LIN {X 0,Y 316.614,Z 405.184,A -85,B 0,C 180,E1 -15553.1,E2 -15553.1} C_VEL
LIN {X 0,Y 315.865,Z 416.609,A -85,B 0,C 180,E1 -15553.852,E2 -15553.852} C_VEL
LIN {X 0,Y 315.165,Z 425.435,A -85,B 0,C 180,E1 -15554.645,E2 -15554.645} C_VEL
LIN {X 0,Y 314.376,Z 433.849,A -85,B 0,C 180,E1 -15555.6,E2 -15555.6} C_VEL
LIN {X 0,Y 313.605,Z 441.806,A -85,B 0,C 180,E1 -15556.721,E2 -15556.721} C_VEL
LIN {X 0,Y 312.821,Z 449.237,A -85,B 0,C 180,E1 -15558.006,E2 -15558.006} C_VEL
LIN {X 0,Y 311.997,Z 456.768,A -85,B 0,C 180,E1 -15559.618,E2 -15559.618} C_VEL
LIN {X 0,Y 311.335,Z 463.636,A -85,B 0,C 180,E1 -15561.563,E2 -15561.563} C_VEL
LIN {X 0,Y 310.91,Z 468.838,A -85,B 0,C 180,E1 -15563.511,E2 -15563.511} C_VEL
LIN {X 0,Y 310.745,Z 472.647,A -85,B 0,C 180,E1 -15565.46,E2 -15565.46} C_VEL
LIN {X 0,Y 310.69,Z 475.122,A -85,B 0,C 180,E1 -15567.407,E2 -15567.407} C_VEL
LIN {X 0,Y 310.648,Z 476.084,A -85,B 0,C 180,E1 -15568.704,E2 -15568.704} C_VEL
LIN {X 0,Y 310.689,Z 476.502,A -85,B 0,C 180,E1 -15570,E2 -15570} C_VEL
LIN {X 0,Y 310.647,Z 476.448,A -85,B 0,C 180,E1 -15571.296,E2 -15571.296} C_VEL
LIN {X 0,Y 310.688,Z 475.928,A -85,B 0,C 180,E1 -15572.593,E2 -15572.593} C_VEL
LIN {X 0,Y 310.749,Z 474.907,A -85,B 0,C 180,E1 -15573.89,E2 -15573.89} C_VEL
LIN {X 0,Y 310.838,Z 472.302,A -85,B 0,C 180,E1 -15575.828,E2 -15575.828} C_VEL
LIN {X 0,Y 311.1,Z 469.9,A -85,B 0,C 180,E1 -15577.137,E2 -15577.137} C_VEL
LIN {X 0,Y 311.63,Z 465.034,A -85,B 0,C 180,E1 -15579.083,E2 -15579.083} C_VEL
LIN {X 0,Y 312.265,Z 459.797,A -85,B 0,C 180,E1 -15580.7,E2 -15580.7} C_VEL
LIN {X 0,Y 313.245,Z 453.258,A -85,B 0,C 180,E1 -15582.306,E2 -15582.306} C_VEL
LIN {X 0,Y 314.329,Z 445.108,A -85,B 0,C 180,E1 -15583.907,E2 -15583.907} C_VEL
LIN {X 0,Y 315.586,Z 435.56,A -85,B 0,C 180,E1 -15585.334,E2 -15585.334} C_VEL
LIN {X 0,Y 316.548,Z 427.654,A -85,B 0,C 180,E1 -15586.278,E2 -15586.278} C_VEL
LIN {X 0,Y 317.389,Z 419.536,A -85,B 0,C 180,E1 -15587.061,E2 -15587.061} C_VEL
LIN {X 0,Y 318.104,Z 411.379,A -85,B 0,C 180,E1 -15587.684,E2 -15587.684} C_VEL
LIN {X 0,Y 318.823,Z 401.925,A -85,B 0,C 180,E1 -15588.221,E2 -15588.221} C_VEL
LIN {X 0,Y 319.332,Z 392.463,A -85,B 0,C 180,E1 -15588.585,E2 -15588.585} C_VEL
LIN {X 0,Y 320.087,Z 349.277,A -85,B 0,C 180,E1 -15589.636,E2 -15589.636} C_VEL
LIN {X 0,Y 316.6,Z 326.517,A -85,B 0,C 180,E1 -15590.471,E2 -15590.471} C_VEL
LIN {X 0,Y 314.474,Z 315.593,A -85,B 0,C 180,E1 -15590.951,E2 -15590.951} C_VEL
LIN {X 0,Y 315.369,Z 306.754,A -85,B 0,C 180,E1 -15593.648,E2 -15593.648} C_VEL
LIN {X 0,Y 314.358,Z 300.169,A -85,B 0,C 180,E1 -15595.831,E2 -15595.831} C_VEL
LIN {X 0,Y 312.514,Z 291.37,A -85,B 0,C 180,E1 -15598.922,E2 -15598.922} C_VEL
LIN {X 0,Y 312.497,Z 291.374,A -85,B 0,C 180,E1 -15602.666,E2 -15602.666} C_VEL
LIN {X 0,Y 312.531,Z 291.369,A -85,B 0,C 180,E1 -15605.949,E2 -15605.949} C_VEL
LIN {X 0,Y 312.499,Z 291.376,A -85,B 0,C 180,E1 -15610.125,E2 -15610.125} C_VEL
LIN {X 0,Y 312.452,Z 291.381,A -85,B 0,C 180,E1 -15613.964,E2 -15613.964} C_VEL
LIN {X 0,Y 312.478,Z 291.372,A -85,B 0,C 180,E1 -15617.918,E2 -15617.918} C_VEL
LIN {X 0,Y 312.496,Z 291.372,A -85,B 0,C 180,E1 -15620.971,E2 -15620.971} C_VEL
LIN {X 0,Y 312.524,Z 291.367,A -85,B 0,C 180,E1 -15624.219,E2 -15624.219} C_VEL
LIN {X 0,Y 312.497,Z 291.363,A -85,B 0,C 180,E1 -15627.333,E2 -15627.333} C_VEL
LIN {X 0,Y 312.544,Z 291.363,A -85,B 0,C 180,E1 -15631.276,E2 -15631.276} C_VEL
LIN {X 0,Y 312.576,Z 291.359,A -85,B 0,C 180,E1 -15634.71,E2 -15634.71} C_VEL
LIN {X 0,Y 312.527,Z 291.357,A -85,B 0,C 180,E1 -15638.912,E2 -15638.912} C_VEL
LIN {X 0,Y 312.629,Z 291.354,A -85,B 0,C 180,E1 -15641.656,E2 -15641.656} C_VEL
LIN {X 0,Y 312.684,Z 291.339,A -85,B 0,C 180,E1 -15645.686,E2 -15645.686} C_VEL
LIN {X 0,Y 312.688,Z 291.339,A -85,B 0,C 180,E1 -15649.642,E2 -15649.642} C_VEL
LIN {X 0,Y 312.843,Z 291.319,A -85,B 0,C 180,E1 -15652.254,E2 -15652.254} C_VEL
LIN {X 0,Y 312.703,Z 291.34,A -85,B 0,C 180,E1 -15654.842,E2 -15654.842} C_VEL
LIN {X 0,Y 312.979,Z 291.306,A -85,B 0,C 180,E1 -15658.713,E2 -15658.713} C_VEL
LIN {X 0,Y 312.98,Z 291.301,A -85,B 0,C 180,E1 -15661.287,E2 -15661.287} C_VEL
LIN {X 0,Y 312.695,Z 291.348,A -85,B 0,C 180,E1 -15665.158,E2 -15665.158} C_VEL
LIN {X 0,Y 312.792,Z 291.324,A -85,B 0,C 180,E1 -15667.748,E2 -15667.748} C_VEL
LIN {X 0,Y 312.659,Z 291.344,A -85,B 0,C 180,E1 -15671.672,E2 -15671.672} C_VEL
LIN {X 0,Y 312.691,Z 291.348,A -85,B 0,C 180,E1 -15674.888,E2 -15674.888} C_VEL
LIN {X 0,Y 312.621,Z 291.36,A -85,B 0,C 180,E1 -15679.237,E2 -15679.237} C_VEL
LIN {X 0,Y 312.538,Z 291.368,A -85,B 0,C 180,E1 -15682.79,E2 -15682.79} C_VEL
LIN {X 0,Y 312.595,Z 291.36,A -85,B 0,C 180,E1 -15685.936,E2 -15685.936} C_VEL
LIN {X 0,Y 312.538,Z 291.366,A -85,B 0,C 180,E1 -15689.651,E2 -15689.651} C_VEL
LIN {X 0,Y 312.513,Z 291.372,A -85,B 0,C 180,E1 -15693.69,E2 -15693.69} C_VEL
LIN {X 0,Y 312.575,Z 291.364,A -85,B 0,C 180,E1 -15697.741,E2 -15697.741} C_VEL
LIN {X 0,Y 312.587,Z 291.595,A -85,B 0,C 180,E1 -15698.104,E2 -15698.104} C_VEL
LIN {X 0,Y 314.358,Z 300.158,A -85,B 0,C 180,E1 -15701.104,E2 -15701.104} C_VEL
LIN {X 0,Y 317.012,Z 307.823,A -85,B 0,C 180,E1 -15701.53,E2 -15701.53} C_VEL
LIN {X 0,Y 320.69,Z 326.341,A -85,B 0,C 180,E1 -15702.278,E2 -15702.278} C_VEL
LIN {X 0,Y 319.477,Z 377.531,A -85,B 0,C 180,E1 -15703.511,E2 -15703.511} C_VEL
LIN {X 0,Y 318.939,Z 388.047,A -85,B 0,C 180,E1 -15703.952,E2 -15703.952} C_VEL
LIN {X 0,Y 318.259,Z 399.5,A -85,B 0,C 180,E1 -15704.703,E2 -15704.703} C_VEL
LIN {X 0,Y 317.369,Z 408.898,A -85,B 0,C 180,E1 -15705.549,E2 -15705.549} C_VEL
LIN {X 0,Y 316.493,Z 417.2,A -85,B 0,C 180,E1 -15706.5,E2 -15706.5} C_VEL
LIN {X 0,Y 315.629,Z 424.127,A -85,B 0,C 180,E1 -15707.465,E2 -15707.465} C_VEL
LIN {X 0,Y 314.701,Z 430.774,A -85,B 0,C 180,E1 -15708.58,E2 -15708.58} C_VEL
LIN {X 0,Y 313.776,Z 437.342,A -85,B 0,C 180,E1 -15709.925,E2 -15709.925} C_VEL
LIN {X 0,Y 313.144,Z 441.993,A -85,B 0,C 180,E1 -15711.068,E2 -15711.068} C_VEL
LIN {X 0,Y 312.365,Z 447.101,A -85,B 0,C 180,E1 -15712.594,E2 -15712.594} C_VEL
LIN {X 0,Y 311.798,Z 451.176,A -85,B 0,C 180,E1 -15714.124,E2 -15714.124} C_VEL
LIN {X 0,Y 311.31,Z 454.327,A -85,B 0,C 180,E1 -15715.641,E2 -15715.641} C_VEL
LIN {X 0,Y 311.064,Z 456.676,A -85,B 0,C 180,E1 -15717.165,E2 -15717.165} C_VEL
LIN {X 0,Y 310.646,Z 458.729,A -85,B 0,C 180,E1 -15719.284,E2 -15719.284} C_VEL
LIN {X 0,Y 310.448,Z 459.46,A -85,B 0,C 180,E1 -15721.615,E2 -15721.615} C_VEL
LIN {X 0,Y 310.449,Z 459.064,A -85,B 0,C 180,E1 -15723.08,E2 -15723.08} C_VEL
LIN {X 0,Y 310.596,Z 457.727,A -85,B 0,C 180,E1 -15724.837,E2 -15724.837} C_VEL
LIN {X 0,Y 310.899,Z 455.22,A -85,B 0,C 180,E1 -15726.698,E2 -15726.698} C_VEL
LIN {X 0,Y 311.215,Z 452.076,A -85,B 0,C 180,E1 -15728.332,E2 -15728.332} C_VEL
LIN {X 0,Y 311.607,Z 448.166,A -85,B 0,C 180,E1 -15729.883,E2 -15729.883} C_VEL
LIN {X 0,Y 312.175,Z 442.501,A -85,B 0,C 180,E1 -15731.629,E2 -15731.629} C_VEL
LIN {X 0,Y 312.802,Z 436.87,A -85,B 0,C 180,E1 -15733.018,E2 -15733.018} C_VEL
LIN {X 0,Y 313.534,Z 430.031,A -85,B 0,C 180,E1 -15734.397,E2 -15734.397} C_VEL
LIN {X 0,Y 314.41,Z 421.641,A -85,B 0,C 180,E1 -15735.766,E2 -15735.766} C_VEL
LIN {X 0,Y 315.327,Z 412.215,A -85,B 0,C 180,E1 -15736.958,E2 -15736.958} C_VEL
LIN {X 0,Y 316.046,Z 403.63,A -85,B 0,C 180,E1 -15737.814,E2 -15737.814} C_VEL
LIN {X 0,Y 316.594,Z 394.035,A -85,B 0,C 180,E1 -15738.557,E2 -15738.557} C_VEL
LIN {X 0,Y 317.053,Z 384.456,A -85,B 0,C 180,E1 -15739.1,E2 -15739.1} C_VEL
LIN {X 0,Y 317.454,Z 374.313,A -85,B 0,C 180,E1 -15739.477,E2 -15739.477} C_VEL
LIN {X 0,Y 318.284,Z 325.044,A -85,B 0,C 180,E1 -15740.639,E2 -15740.639} C_VEL
LIN {X 0,Y 313.875,Z 300.254,A -85,B 0,C 180,E1 -15741.51,E2 -15741.51} C_VEL
LIN {X 0,Y 313.394,Z 294.514,A -85,B 0,C 180,E1 -15743.562,E2 -15743.562} C_VEL
LIN {X 0,Y 312.735,Z 291.343,A -85,B 0,C 180,E1 -15744.762,E2 -15744.762} C_VEL
LIN {X 0,Y 312.99,Z 291.307,A -85,B 0,C 180,E1 -15748.713,E2 -15748.713} C_VEL
LIN {X 0,Y 312.991,Z 291.307,A -85,B 0,C 180,E1 -15751.287,E2 -15751.287} C_VEL
LIN {X 0,Y 312.709,Z 291.341,A -85,B 0,C 180,E1 -15755.158,E2 -15755.158} C_VEL
LIN {X 0,Y 312.82,Z 291.33,A -85,B 0,C 180,E1 -15757.747,E2 -15757.747} C_VEL
LIN {X 0,Y 312.671,Z 291.346,A -85,B 0,C 180,E1 -15761.671,E2 -15761.671} C_VEL
LIN {X 0,Y 312.668,Z 291.349,A -85,B 0,C 180,E1 -15764.865,E2 -15764.865} C_VEL
LIN {X 0,Y 312.586,Z 291.357,A -85,B 0,C 180,E1 -15769.212,E2 -15769.212} C_VEL
LIN {X 0,Y 312.526,Z 291.369,A -85,B 0,C 180,E1 -15772.78,E2 -15772.78} C_VEL
LIN {X 0,Y 312.596,Z 291.356,A -85,B 0,C 180,E1 -15775.933,E2 -15775.933} C_VEL
LIN {X 0,Y 312.544,Z 291.363,A -85,B 0,C 180,E1 -15779.649,E2 -15779.649} C_VEL
LIN {X 0,Y 312.517,Z 291.366,A -85,B 0,C 180,E1 -15783.688,E2 -15783.688} C_VEL
LIN {X 0,Y 312.517,Z 291.37,A -85,B 0,C 180,E1 -15787.385,E2 -15787.385} C_VEL
LIN {X 0,Y 312.487,Z 291.369,A -85,B 0,C 180,E1 -15790.708,E2 -15790.708} C_VEL
LIN {X 0,Y 312.506,Z 291.367,A -85,B 0,C 180,E1 -15794.198,E2 -15794.198} C_VEL
LIN {X 0,Y 312.544,Z 291.365,A -85,B 0,C 180,E1 -15797.905,E2 -15797.905} C_VEL
LIN {X 0,Y 312.538,Z 291.366,A -85,B 0,C 180,E1 -15801.907,E2 -15801.907} C_VEL
LIN {X 0,Y 312.5,Z 291.37,A -85,B 0,C 180,E1 -15805.789,E2 -15805.789} C_VEL
LIN {X 0,Y 312.502,Z 291.369,A -85,B 0,C 180,E1 -15805.999,E2 -15805.999} C_VEL
LIN {X 0,Y 311.861,Z 291.447,A -85,B 0,C 180,E1 -15807.075,E2 -15807.075} C_VEL
LIN {X 0,Y 309.03,Z 291.799,A -85,B 0,C 180,E1 -15808.827,E2 -15808.827} C_VEL
LIN {X 0,Y 306.614,Z 292.105,A -85,B 0,C 180,E1 -15810.247,E2 -15810.247} C_VEL
LIN {X 0,Y 305.574,Z 292.231,A -85,B 0,C 180,E1 -15811.347,E2 -15811.347} C_VEL
LIN {X 0,Y 305.489,Z 292.238,A -85,B 0,C 180,E1 -15811.72,E2 -15811.72} C_VEL
LIN {X 0,Y 305.564,Z 292.236,A -85,B 0,C 180,E1 -15814.087,E2 -15814.087} C_VEL
LIN {X 0,Y 305.492,Z 292.242,A -85,B 0,C 180,E1 -15818.402,E2 -15818.402} C_VEL
LIN {X 0,Y 305.582,Z 292.228,A -85,B 0,C 180,E1 -15821.217,E2 -15821.217} C_VEL
LIN {X 0,Y 305.64,Z 292.222,A -85,B 0,C 180,E1 -15825.348,E2 -15825.348} C_VEL
LIN {X 0,Y 305.626,Z 292.224,A -85,B 0,C 180,E1 -15829.399,E2 -15829.399} C_VEL
LIN {X 0,Y 305.787,Z 292.203,A -85,B 0,C 180,E1 -15832.074,E2 -15832.074} C_VEL
LIN {X 0,Y 305.676,Z 292.219,A -85,B 0,C 180,E1 -15834.723,E2 -15834.723} C_VEL
LIN {X 0,Y 305.947,Z 292.185,A -85,B 0,C 180,E1 -15838.684,E2 -15838.684} C_VEL
LIN {X 0,Y 305.949,Z 292.188,A -85,B 0,C 180,E1 -15841.316,E2 -15841.316} C_VEL
LIN {X 0,Y 305.832,Z 292.198,A -85,B 0,C 180,E1 -15846.598,E2 -15846.598} C_VEL
LIN {X 0,Y 305.696,Z 292.217,A -85,B 0,C 180,E1 -15849.261,E2 -15849.261} C_VEL
LIN {X 0,Y 305.581,Z 292.232,A -85,B 0,C 180,E1 -15853.296,E2 -15853.296} C_VEL
LIN {X 0,Y 305.585,Z 292.232,A -85,B 0,C 180,E1 -15856.02,E2 -15856.02} C_VEL
LIN {X 0,Y 305.552,Z 292.235,A -85,B 0,C 180,E1 -15859.436,E2 -15859.436} C_VEL
LIN {X 0,Y 305.478,Z 292.241,A -85,B 0,C 180,E1 -15863.04,E2 -15863.04} C_VEL
LIN {X 0,Y 305.523,Z 292.241,A -85,B 0,C 180,E1 -15866.221,E2 -15866.221} C_VEL
LIN {X 0,Y 305.48,Z 292.241,A -85,B 0,C 180,E1 -15869.048,E2 -15869.048} C_VEL
LIN {X 0,Y 305.434,Z 292.25,A -85,B 0,C 180,E1 -15871.953,E2 -15871.953} C_VEL
LIN {X 0,Y 305.455,Z 292.246,A -85,B 0,C 180,E1 -15875.114,E2 -15875.114} C_VEL
LIN {X 0,Y 305.442,Z 292.25,A -85,B 0,C 180,E1 -15878.529,E2 -15878.529} C_VEL
LIN {X 0,Y 305.453,Z 292.248,A -85,B 0,C 180,E1 -15882.587,E2 -15882.587} C_VEL
LIN {X 0,Y 305.437,Z 292.25,A -85,B 0,C 180,E1 -15886.349,E2 -15886.349} C_VEL
LIN {X 0,Y 305.453,Z 292.245,A -85,B 0,C 180,E1 -15889.893,E2 -15889.893} C_VEL
LIN {X 0,Y 305.476,Z 292.244,A -85,B 0,C 180,E1 -15893.633,E2 -15893.633} C_VEL
LIN {X 0,Y 305.461,Z 292.245,A -85,B 0,C 180,E1 -15896.484,E2 -15896.484} C_VEL
LIN {X 0,Y 305.428,Z 292.252,A -85,B 0,C 180,E1 -15899.588,E2 -15899.588} C_VEL
LIN {X 0,Y 305.523,Z 292.28,A -85,B 0,C 180,E1 -15902.052,E2 -15902.052} C_VEL
LIN {X 0,Y 307.662,Z 303.716,A -85,B 0,C 180,E1 -15906.026,E2 -15906.026} C_VEL
LIN {X 0,Y 307.694,Z 307.146,A -85,B 0,C 180,E1 -15907.152,E2 -15907.152} C_VEL
LIN {X 0,Y 306.626,Z 316.497,A -85,B 0,C 180,E1 -15910.125,E2 -15910.125} C_VEL
LIN {X 0,Y 311.183,Z 350.857,A -85,B 0,C 180,E1 -15911.24,E2 -15911.24} C_VEL
LIN {X 0,Y 310.4,Z 393.592,A -85,B 0,C 180,E1 -15912.292,E2 -15912.292} C_VEL
LIN {X 0,Y 309.872,Z 403.563,A -85,B 0,C 180,E1 -15912.705,E2 -15912.705} C_VEL
LIN {X 0,Y 309.112,Z 414.767,A -85,B 0,C 180,E1 -15913.404,E2 -15913.404} C_VEL
LIN {X 0,Y 308.293,Z 424.721,A -85,B 0,C 180,E1 -15914.294,E2 -15914.294} C_VEL
LIN {X 0,Y 307.452,Z 433.226,A -85,B 0,C 180,E1 -15915.268,E2 -15915.268} C_VEL
LIN {X 0,Y 306.613,Z 441.254,A -85,B 0,C 180,E1 -15916.412,E2 -15916.412} C_VEL
LIN {X 0,Y 306.013,Z 447.028,A -85,B 0,C 180,E1 -15917.398,E2 -15917.398} C_VEL
LIN {X 0,Y 305.307,Z 453.471,A -85,B 0,C 180,E1 -15918.717,E2 -15918.717} C_VEL
LIN {X 0,Y 304.738,Z 458.821,A -85,B 0,C 180,E1 -15920.04,E2 -15920.04} C_VEL
LIN {X 0,Y 304.306,Z 463.278,A -85,B 0,C 180,E1 -15921.366,E2 -15921.366} C_VEL
LIN {X 0,Y 303.844,Z 468.514,A -85,B 0,C 180,E1 -15923.359,E2 -15923.359} C_VEL
LIN {X 0,Y 303.651,Z 472.353,A -85,B 0,C 180,E1 -15925.354,E2 -15925.354} C_VEL
LIN {X 0,Y 303.615,Z 474.879,A -85,B 0,C 180,E1 -15927.347,E2 -15927.347} C_VEL
LIN {X 0,Y 303.566,Z 475.848,A -85,B 0,C 180,E1 -15928.673,E2 -15928.673} C_VEL
LIN {X 0,Y 303.601,Z 476.291,A -85,B 0,C 180,E1 -15930,E2 -15930} C_VEL
LIN {X 0,Y 303.565,Z 476.263,A -85,B 0,C 180,E1 -15931.327,E2 -15931.327} C_VEL
LIN {X 0,Y 303.614,Z 475.769,A -85,B 0,C 180,E1 -15932.653,E2 -15932.653} C_VEL
LIN {X 0,Y 303.665,Z 474.758,A -85,B 0,C 180,E1 -15933.981,E2 -15933.981} C_VEL
LIN {X 0,Y 303.73,Z 472.564,A -85,B 0,C 180,E1 -15935.747,E2 -15935.747} C_VEL
LIN {X 0,Y 304.046,Z 469.815,A -85,B 0,C 180,E1 -15937.304,E2 -15937.304} C_VEL
LIN {X 0,Y 304.618,Z 465.004,A -85,B 0,C 180,E1 -15939.294,E2 -15939.294} C_VEL
LIN {X 0,Y 305.284,Z 459.813,A -85,B 0,C 180,E1 -15940.948,E2 -15940.948} C_VEL
LIN {X 0,Y 306.076,Z 454.747,A -85,B 0,C 180,E1 -15942.262,E2 -15942.262} C_VEL
LIN {X 0,Y 306.992,Z 448.655,A -85,B 0,C 180,E1 -15943.571,E2 -15943.571} C_VEL
LIN {X 0,Y 307.963,Z 441.26,A -85,B 0,C 180,E1 -15944.876,E2 -15944.876} C_VEL
LIN {X 0,Y 309.083,Z 433.349,A -85,B 0,C 180,E1 -15946.003,E2 -15946.003} C_VEL
LIN {X 0,Y 310.326,Z 423.508,A -85,B 0,C 180,E1 -15947.122,E2 -15947.122} C_VEL
LIN {X 0,Y 311.38,Z 412.054,A -85,B 0,C 180,E1 -15948.079,E2 -15948.079} C_VEL
LIN {X 0,Y 312.138,Z 402.465,A -85,B 0,C 180,E1 -15948.649,E2 -15948.649} C_VEL
LIN {X 0,Y 312.702,Z 392.836,A -85,B 0,C 180,E1 -15949.037,E2 -15949.037} C_VEL
LIN {X 0,Y 313.516,Z 350.323,A -85,B 0,C 180,E1 -15950.099,E2 -15950.099} C_VEL
LIN {X 0,Y 310.134,Z 327.944,A -85,B 0,C 180,E1 -15950.947,E2 -15950.947} C_VEL
LIN {X 0,Y 307.65,Z 315.355,A -85,B 0,C 180,E1 -15951.526,E2 -15951.526} C_VEL
LIN {X 0,Y 308.449,Z 307.895,A -85,B 0,C 180,E1 -15953.855,E2 -15953.855} C_VEL
LIN {X 0,Y 307.261,Z 300.885,A -85,B 0,C 180,E1 -15956.247,E2 -15956.247} C_VEL
LIN {X 0,Y 305.468,Z 292.248,A -85,B 0,C 180,E1 -15959.379,E2 -15959.379} C_VEL
LIN {X 0,Y 305.461,Z 292.248,A -85,B 0,C 180,E1 -15963.516,E2 -15963.516} C_VEL
LIN {X 0,Y 305.471,Z 292.249,A -85,B 0,C 180,E1 -15966.739,E2 -15966.739} C_VEL
LIN {X 0,Y 305.45,Z 292.256,A -85,B 0,C 180,E1 -15970.599,E2 -15970.599} C_VEL
LIN {X 0,Y 305.42,Z 292.259,A -85,B 0,C 180,E1 -15973.654,E2 -15973.654} C_VEL
LIN {X 0,Y 305.449,Z 292.252,A -85,B 0,C 180,E1 -15977.414,E2 -15977.414} C_VEL
LIN {X 0,Y 305.469,Z 292.244,A -85,B 0,C 180,E1 -15981.597,E2 -15981.597} C_VEL
LIN {X 0,Y 305.455,Z 292.247,A -85,B 0,C 180,E1 -15984.886,E2 -15984.886} C_VEL
LIN {X 0,Y 305.444,Z 292.245,A -85,B 0,C 180,E1 -15988.354,E2 -15988.354} C_VEL
LIN {X 0,Y 305.512,Z 292.238,A -85,B 0,C 180,E1 -15991.113,E2 -15991.113} C_VEL
LIN {X 0,Y 305.563,Z 292.229,A -85,B 0,C 180,E1 -15994.087,E2 -15994.087} C_VEL
LIN {X 0,Y 305.472,Z 292.233,A -85,B 0,C 180,E1 -15998.401,E2 -15998.401} C_VEL
LIN {X 0,Y 305.58,Z 292.231,A -85,B 0,C 180,E1 -16001.217,E2 -16001.217} C_VEL
LIN {X 0,Y 305.64,Z 292.216,A -85,B 0,C 180,E1 -16005.349,E2 -16005.349} C_VEL
LIN {X 0,Y 305.626,Z 292.218,A -85,B 0,C 180,E1 -16009.399,E2 -16009.399} C_VEL
LIN {X 0,Y 305.787,Z 292.197,A -85,B 0,C 180,E1 -16012.074,E2 -16012.074} C_VEL
LIN {X 0,Y 305.675,Z 292.217,A -85,B 0,C 180,E1 -16014.723,E2 -16014.723} C_VEL
LIN {X 0,Y 305.946,Z 292.182,A -85,B 0,C 180,E1 -16018.684,E2 -16018.684} C_VEL
LIN {X 0,Y 305.946,Z 292.176,A -85,B 0,C 180,E1 -16021.316,E2 -16021.316} C_VEL
LIN {X 0,Y 305.664,Z 292.223,A -85,B 0,C 180,E1 -16025.277,E2 -16025.277} C_VEL
LIN {X 0,Y 305.741,Z 292.203,A -85,B 0,C 180,E1 -16027.928,E2 -16027.928} C_VEL
LIN {X 0,Y 305.593,Z 292.222,A -85,B 0,C 180,E1 -16031.946,E2 -16031.946} C_VEL
LIN {X 0,Y 305.629,Z 292.228,A -85,B 0,C 180,E1 -16035.035,E2 -16035.035} C_VEL
LIN {X 0,Y 305.568,Z 292.237,A -85,B 0,C 180,E1 -16039.445,E2 -16039.445} C_VEL
LIN {X 0,Y 305.483,Z 292.248,A -85,B 0,C 180,E1 -16043.042,E2 -16043.042} C_VEL
LIN {X 0,Y 305.54,Z 292.237,A -85,B 0,C 180,E1 -16046.228,E2 -16046.228} C_VEL
LIN {X 0,Y 305.488,Z 292.241,A -85,B 0,C 180,E1 -16049.051,E2 -16049.051} C_VEL
LIN {X 0,Y 305.438,Z 292.254,A -85,B 0,C 180,E1 -16051.953,E2 -16051.953} C_VEL
LIN {X 0,Y 305.456,Z 292.243,A -85,B 0,C 180,E1 -16055.114,E2 -16055.114} C_VEL
LIN {X 0,Y 305.537,Z 292.337,A -85,B 0,C 180,E1 -16057.61,E2 -16057.61} C_VEL
LIN {X 0,Y 307.281,Z 300.534,A -85,B 0,C 180,E1 -16060.533,E2 -16060.533} C_VEL
LIN {X 0,Y 310.625,Z 309.688,A -85,B 0,C 180,E1 -16061.06,E2 -16061.06} C_VEL
LIN {X 0,Y 314.1,Z 327.127,A -85,B 0,C 180,E1 -16061.797,E2 -16061.797} C_VEL
LIN {X 0,Y 312.86,Z 377.956,A -85,B 0,C 180,E1 -16063.051,E2 -16063.051} C_VEL
LIN {X 0,Y 312.294,Z 388.928,A -85,B 0,C 180,E1 -16063.528,E2 -16063.528} C_VEL
LIN {X 0,Y 311.562,Z 400.101,A -85,B 0,C 180,E1 -16064.293,E2 -16064.293} C_VEL
LIN {X 0,Y 310.726,Z 408.69,A -85,B 0,C 180,E1 -16065.078,E2 -16065.078} C_VEL
LIN {X 0,Y 309.738,Z 417.464,A -85,B 0,C 180,E1 -16066.099,E2 -16066.099} C_VEL
LIN {X 0,Y 308.77,Z 424.848,A -85,B 0,C 180,E1 -16067.159,E2 -16067.159} C_VEL
LIN {X 0,Y 307.792,Z 431.512,A -85,B 0,C 180,E1 -16068.317,E2 -16068.317} C_VEL
LIN {X 0,Y 306.807,Z 438.088,A -85,B 0,C 180,E1 -16069.713,E2 -16069.713} C_VEL
LIN {X 0,Y 305.904,Z 444.354,A -85,B 0,C 180,E1 -16071.365,E2 -16071.365} C_VEL
LIN {X 0,Y 305.064,Z 449.819,A -85,B 0,C 180,E1 -16073.204,E2 -16073.204} C_VEL
LIN {X 0,Y 304.435,Z 453.337,A -85,B 0,C 180,E1 -16074.752,E2 -16074.752} C_VEL
LIN {X 0,Y 304.109,Z 456.025,A -85,B 0,C 180,E1 -16076.315,E2 -16076.315} C_VEL
LIN {X 0,Y 303.822,Z 457.919,A -85,B 0,C 180,E1 -16077.858,E2 -16077.858} C_VEL
LIN {X 0,Y 303.537,Z 459.083,A -85,B 0,C 180,E1 -16079.378,E2 -16079.378} C_VEL
LIN {X 0,Y 303.35,Z 459.626,A -85,B 0,C 180,E1 -16081.689,E2 -16081.689} C_VEL
LIN {X 0,Y 303.476,Z 458.165,A -85,B 0,C 180,E1 -16084.579,E2 -16084.579} C_VEL
LIN {X 0,Y 303.826,Z 455.253,A -85,B 0,C 180,E1 -16086.845,E2 -16086.845} C_VEL
LIN {X 0,Y 304.113,Z 452.558,A -85,B 0,C 180,E1 -16088.3,E2 -16088.3} C_VEL
LIN {X 0,Y 304.478,Z 449.135,A -85,B 0,C 180,E1 -16089.744,E2 -16089.744} C_VEL
LIN {X 0,Y 305.034,Z 443.643,A -85,B 0,C 180,E1 -16091.531,E2 -16091.531} C_VEL
LIN {X 0,Y 305.668,Z 438.202,A -85,B 0,C 180,E1 -16092.954,E2 -16092.954} C_VEL
LIN {X 0,Y 306.424,Z 431.257,A -85,B 0,C 180,E1 -16094.428,E2 -16094.428} C_VEL
LIN {X 0,Y 307.302,Z 423.453,A -85,B 0,C 180,E1 -16095.768,E2 -16095.768} C_VEL
LIN {X 0,Y 308.335,Z 413.384,A -85,B 0,C 180,E1 -16097.137,E2 -16097.137} C_VEL
LIN {X 0,Y 309.206,Z 402.906,A -85,B 0,C 180,E1 -16098.196,E2 -16098.196} C_VEL
LIN {X 0,Y 309.715,Z 394.179,A -85,B 0,C 180,E1 -16098.879,E2 -16098.879} C_VEL
LIN {X 0,Y 310.2,Z 384.57,A -85,B 0,C 180,E1 -16099.434,E2 -16099.434} C_VEL
LIN {X 0,Y 310.626,Z 374.363,A -85,B 0,C 180,E1 -16099.819,E2 -16099.819} C_VEL
LIN {X 0,Y 311.438,Z 325.729,A -85,B 0,C 180,E1 -16100.993,E2 -16100.993} C_VEL
LIN {X 0,Y 306.889,Z 300.481,A -85,B 0,C 180,E1 -16101.896,E2 -16101.896} C_VEL
LIN {X 0,Y 306.224,Z 294.539,A -85,B 0,C 180,E1 -16104.072,E2 -16104.072} C_VEL
LIN {X 0,Y 305.671,Z 292.223,A -85,B 0,C 180,E1 -16104.971,E2 -16104.971} C_VEL
LIN {X 0,Y 305.957,Z 292.184,A -85,B 0,C 180,E1 -16108.684,E2 -16108.684} C_VEL
LIN {X 0,Y 305.957,Z 292.184,A -85,B 0,C 180,E1 -16111.316,E2 -16111.316} C_VEL
LIN {X 0,Y 305.678,Z 292.217,A -85,B 0,C 180,E1 -16115.277,E2 -16115.277} C_VEL
LIN {X 0,Y 305.766,Z 292.21,A -85,B 0,C 180,E1 -16117.927,E2 -16117.927} C_VEL
LIN {X 0,Y 305.605,Z 292.228,A -85,B 0,C 180,E1 -16121.945,E2 -16121.945} C_VEL
LIN {X 0,Y 305.61,Z 292.227,A -85,B 0,C 180,E1 -16125.014,E2 -16125.014} C_VEL
LIN {X 0,Y 305.542,Z 292.233,A -85,B 0,C 180,E1 -16129.426,E2 -16129.426} C_VEL
LIN {X 0,Y 305.486,Z 292.243,A -85,B 0,C 180,E1 -16133.039,E2 -16133.039} C_VEL
LIN {X 0,Y 305.526,Z 292.237,A -85,B 0,C 180,E1 -16136.218,E2 -16136.218} C_VEL
LIN {X 0,Y 305.495,Z 292.246,A -85,B 0,C 180,E1 -16139.049,E2 -16139.049} C_VEL
LIN {X 0,Y 305.463,Z 292.246,A -85,B 0,C 180,E1 -16143.516,E2 -16143.516} C_VEL
LIN {X 0,Y 305.47,Z 292.245,A -85,B 0,C 180,E1 -16146.739,E2 -16146.739} C_VEL
LIN {X 0,Y 305.452,Z 292.245,A -85,B 0,C 180,E1 -16150.599,E2 -16150.599} C_VEL
LIN {X 0,Y 305.451,Z 292.245,A -85,B 0,C 180,E1 -16154.498,E2 -16154.498} C_VEL
LIN {X 0,Y 305.49,Z 292.242,A -85,B 0,C 180,E1 -16158.151,E2 -16158.151} C_VEL
LIN {X 0,Y 305.504,Z 292.243,A -85,B 0,C 180,E1 -16161.601,E2 -16161.601} C_VEL
LIN {X 0,Y 305.456,Z 292.242,A -85,B 0,C 180,E1 -16164.886,E2 -16164.886} C_VEL
LIN {X 0,Y 305.446,Z 292.248,A -85,B 0,C 180,E1 -16168.354,E2 -16168.354} C_VEL
LIN {X 0,Y 305.489,Z 292.238,A -85,B 0,C 180,E1 -16171.72,E2 -16171.72} C_VEL
LIN {X 0,Y 304.812,Z 292.326,A -85,B 0,C 180,E1 -16172.82,E2 -16172.82} C_VEL
LIN {X 0,Y 301.934,Z 292.685,A -85,B 0,C 180,E1 -16174.611,E2 -16174.611} C_VEL
LIN {X 0,Y 299.509,Z 292.989,A -85,B 0,C 180,E1 -16176.063,E2 -16176.063} C_VEL
LIN {X 0,Y 298.486,Z 293.111,A -85,B 0,C 180,E1 -16177.189,E2 -16177.189} C_VEL
LIN {X 0,Y 298.412,Z 293.12,A -85,B 0,C 180,E1 -16177.57,E2 -16177.57} C_VEL
LIN {X 0,Y 298.531,Z 293.108,A -85,B 0,C 180,E1 -16180.756,E2 -16180.756} C_VEL
LIN {X 0,Y 298.585,Z 293.103,A -85,B 0,C 180,E1 -16184.994,E2 -16184.994} C_VEL
LIN {X 0,Y 298.582,Z 293.103,A -85,B 0,C 180,E1 -16189.146,E2 -16189.146} C_VEL
LIN {X 0,Y 298.732,Z 293.081,A -85,B 0,C 180,E1 -16191.885,E2 -16191.885} C_VEL
LIN {X 0,Y 298.647,Z 293.092,A -85,B 0,C 180,E1 -16194.599,E2 -16194.599} C_VEL
LIN {X 0,Y 298.914,Z 293.06,A -85,B 0,C 180,E1 -16198.653,E2 -16198.653} C_VEL
LIN {X 0,Y 298.915,Z 293.064,A -85,B 0,C 180,E1 -16201.347,E2 -16201.347} C_VEL
LIN {X 0,Y 298.777,Z 293.077,A -85,B 0,C 180,E1 -16206.754,E2 -16206.754} C_VEL
LIN {X 0,Y 298.628,Z 293.097,A -85,B 0,C 180,E1 -16209.482,E2 -16209.482} C_VEL
LIN {X 0,Y 298.544,Z 293.111,A -85,B 0,C 180,E1 -16213.616,E2 -16213.616} C_VEL
LIN {X 0,Y 298.54,Z 293.107,A -85,B 0,C 180,E1 -16216.409,E2 -16216.409} C_VEL
LIN {X 0,Y 298.489,Z 293.116,A -85,B 0,C 180,E1 -16219.647,E2 -16219.647} C_VEL
LIN {X 0,Y 298.421,Z 293.123,A -85,B 0,C 180,E1 -16223.601,E2 -16223.601} C_VEL
LIN {X 0,Y 298.479,Z 293.116,A -85,B 0,C 180,E1 -16226.575,E2 -16226.575} C_VEL
LIN {X 0,Y 298.409,Z 293.124,A -85,B 0,C 180,E1 -16229.642,E2 -16229.642} C_VEL
LIN {X 0,Y 298.387,Z 293.127,A -85,B 0,C 180,E1 -16232.801,E2 -16232.801} C_VEL
LIN {X 0,Y 298.439,Z 293.121,A -85,B 0,C 180,E1 -16236.808,E2 -16236.808} C_VEL
LIN {X 0,Y 298.381,Z 293.124,A -85,B 0,C 180,E1 -16241.088,E2 -16241.088} C_VEL
LIN {X 0,Y 298.384,Z 293.129,A -85,B 0,C 180,E1 -16245.042,E2 -16245.042} C_VEL
LIN {X 0,Y 298.383,Z 293.132,A -85,B 0,C 180,E1 -16248.913,E2 -16248.913} C_VEL
LIN {X 0,Y 298.44,Z 293.123,A -85,B 0,C 180,E1 -16253.194,E2 -16253.194} C_VEL
LIN {X 0,Y 298.389,Z 293.131,A -85,B 0,C 180,E1 -16257.2,E2 -16257.2} C_VEL
LIN {X 0,Y 298.496,Z 293.222,A -85,B 0,C 180,E1 -16261.813,E2 -16261.813} C_VEL
LIN {X 0,Y 300.574,Z 304.323,A -85,B 0,C 180,E1 -16265.768,E2 -16265.768} C_VEL
LIN {X 0,Y 300.706,Z 307.828,A -85,B 0,C 180,E1 -16266.954,E2 -16266.954} C_VEL
LIN {X 0,Y 299.695,Z 316.38,A -85,B 0,C 180,E1 -16269.721,E2 -16269.721} C_VEL
LIN {X 0,Y 304.355,Z 351.53,A -85,B 0,C 180,E1 -16270.892,E2 -16270.892} C_VEL
LIN {X 0,Y 303.531,Z 393.97,A -85,B 0,C 180,E1 -16271.966,E2 -16271.966} C_VEL
LIN {X 0,Y 302.916,Z 404.928,A -85,B 0,C 180,E1 -16272.446,E2 -16272.446} C_VEL
LIN {X 0,Y 302.045,Z 416.713,A -85,B 0,C 180,E1 -16273.266,E2 -16273.266} C_VEL
LIN {X 0,Y 301.302,Z 425.445,A -85,B 0,C 180,E1 -16274.094,E2 -16274.094} C_VEL
LIN {X 0,Y 300.443,Z 433.787,A -85,B 0,C 180,E1 -16275.09,E2 -16275.09} C_VEL
LIN {X 0,Y 299.573,Z 441.689,A -85,B 0,C 180,E1 -16276.259,E2 -16276.259} C_VEL
LIN {X 0,Y 298.889,Z 448.223,A -85,B 0,C 180,E1 -16277.438,E2 -16277.438} C_VEL
LIN {X 0,Y 298.163,Z 454.435,A -85,B 0,C 180,E1 -16278.787,E2 -16278.787} C_VEL
LIN {X 0,Y 297.596,Z 459.586,A -85,B 0,C 180,E1 -16280.142,E2 -16280.142} C_VEL
LIN {X 0,Y 297.075,Z 464.832,A -85,B 0,C 180,E1 -16281.84,E2 -16281.84} C_VEL
LIN {X 0,Y 296.679,Z 469.69,A -85,B 0,C 180,E1 -16283.881,E2 -16283.881} C_VEL
LIN {X 0,Y 296.563,Z 473.032,A -85,B 0,C 180,E1 -16285.923,E2 -16285.923} C_VEL
LIN {X 0,Y 296.543,Z 474.627,A -85,B 0,C 180,E1 -16287.283,E2 -16287.283} C_VEL
LIN {X 0,Y 296.486,Z 475.607,A -85,B 0,C 180,E1 -16288.642,E2 -16288.642} C_VEL
LIN {X 0,Y 296.516,Z 476.079,A -85,B 0,C 180,E1 -16290,E2 -16290} C_VEL
LIN {X 0,Y 296.485,Z 476.081,A -85,B 0,C 180,E1 -16291.358,E2 -16291.358} C_VEL
LIN {X 0,Y 296.541,Z 475.617,A -85,B 0,C 180,E1 -16292.717,E2 -16292.717} C_VEL
LIN {X 0,Y 296.563,Z 474.614,A -85,B 0,C 180,E1 -16294.077,E2 -16294.077} C_VEL
LIN {X 0,Y 296.622,Z 472.751,A -85,B 0,C 180,E1 -16295.661,E2 -16295.661} C_VEL
LIN {X 0,Y 296.989,Z 469.736,A -85,B 0,C 180,E1 -16297.478,E2 -16297.478} C_VEL
LIN {X 0,Y 297.592,Z 464.984,A -85,B 0,C 180,E1 -16299.515,E2 -16299.515} C_VEL
LIN {X 0,Y 298.321,Z 459.832,A -85,B 0,C 180,E1 -16301.207,E2 -16301.207} C_VEL
LIN {X 0,Y 299.158,Z 454.81,A -85,B 0,C 180,E1 -16302.55,E2 -16302.55} C_VEL
LIN {X 0,Y 300.098,Z 448.769,A -85,B 0,C 180,E1 -16303.889,E2 -16303.889} C_VEL
LIN {X 0,Y 301.126,Z 441.434,A -85,B 0,C 180,E1 -16305.222,E2 -16305.222} C_VEL
LIN {X 0,Y 302.281,Z 433.598,A -85,B 0,C 180,E1 -16306.373,E2 -16306.373} C_VEL
LIN {X 0,Y 303.385,Z 425.351,A -85,B 0,C 180,E1 -16307.352,E2 -16307.352} C_VEL
LIN {X 0,Y 304.416,Z 414.922,A -85,B 0,C 180,E1 -16308.334,E2 -16308.334} C_VEL
LIN {X 0,Y 305.481,Z 403.081,A -85,B 0,C 180,E1 -16309.094,E2 -16309.094} C_VEL
LIN {X 0,Y 306.096,Z 393.634,A -85,B 0,C 180,E1 -16309.497,E2 -16309.497} C_VEL
LIN {X 0,Y 307.054,Z 351.976,A -85,B 0,C 180,E1 -16310.564,E2 -16310.564} C_VEL
LIN {X 0,Y 304.045,Z 331.186,A -85,B 0,C 180,E1 -16311.37,E2 -16311.37} C_VEL
LIN {X 0,Y 300.832,Z 315.256,A -85,B 0,C 180,E1 -16312.084,E2 -16312.084} C_VEL
LIN {X 0,Y 301.534,Z 309.428,A -85,B 0,C 180,E1 -16313.941,E2 -16313.941} C_VEL
LIN {X 0,Y 300.352,Z 302.438,A -85,B 0,C 180,E1 -16316.396,E2 -16316.396} C_VEL
LIN {X 0,Y 298.406,Z 293.131,A -85,B 0,C 180,E1 -16319.836,E2 -16319.836} C_VEL
LIN {X 0,Y 298.389,Z 293.132,A -85,B 0,C 180,E1 -16322.8,E2 -16322.8} C_VEL
LIN {X 0,Y 298.442,Z 293.124,A -85,B 0,C 180,E1 -16326.807,E2 -16326.807} C_VEL
LIN {X 0,Y 298.382,Z 293.137,A -85,B 0,C 180,E1 -16331.087,E2 -16331.087} C_VEL
LIN {X 0,Y 298.394,Z 293.133,A -85,B 0,C 180,E1 -16333.102,E2 -16333.102} C_VEL
LIN {X 0,Y 298.397,Z 293.131,A -85,B 0,C 180,E1 -16336.92,E2 -16336.92} C_VEL
LIN {X 0,Y 298.397,Z 293.128,A -85,B 0,C 180,E1 -16341.006,E2 -16341.006} C_VEL
LIN {X 0,Y 298.411,Z 293.123,A -85,B 0,C 180,E1 -16343.929,E2 -16343.929} C_VEL
LIN {X 0,Y 298.387,Z 293.121,A -85,B 0,C 180,E1 -16347.983,E2 -16347.983} C_VEL
LIN {X 0,Y 298.455,Z 293.11,A -85,B 0,C 180,E1 -16351.904,E2 -16351.904} C_VEL
LIN {X 0,Y 298.475,Z 293.115,A -85,B 0,C 180,E1 -16354.923,E2 -16354.923} C_VEL
LIN {X 0,Y 298.43,Z 293.114,A -85,B 0,C 180,E1 -16359.314,E2 -16359.314} C_VEL
LIN {X 0,Y 298.528,Z 293.11,A -85,B 0,C 180,E1 -16362.179,E2 -16362.179} C_VEL
LIN {X 0,Y 298.584,Z 293.092,A -85,B 0,C 180,E1 -16364.994,E2 -16364.994} C_VEL
LIN {X 0,Y 298.582,Z 293.097,A -85,B 0,C 180,E1 -16369.146,E2 -16369.146} C_VEL
LIN {X 0,Y 298.731,Z 293.075,A -85,B 0,C 180,E1 -16371.885,E2 -16371.885} C_VEL
LIN {X 0,Y 298.646,Z 293.093,A -85,B 0,C 180,E1 -16374.599,E2 -16374.599} C_VEL
LIN {X 0,Y 298.913,Z 293.058,A -85,B 0,C 180,E1 -16378.653,E2 -16378.653} C_VEL
LIN {X 0,Y 298.913,Z 293.052,A -85,B 0,C 180,E1 -16381.347,E2 -16381.347} C_VEL
LIN {X 0,Y 298.632,Z 293.097,A -85,B 0,C 180,E1 -16385.402,E2 -16385.402} C_VEL
LIN {X 0,Y 298.7,Z 293.083,A -85,B 0,C 180,E1 -16388.822,E2 -16388.822} C_VEL
LIN {X 0,Y 298.543,Z 293.099,A -85,B 0,C 180,E1 -16392.232,E2 -16392.232} C_VEL
LIN {X 0,Y 298.577,Z 293.108,A -85,B 0,C 180,E1 -16395.195,E2 -16395.195} C_VEL
LIN {X 0,Y 298.531,Z 293.115,A -85,B 0,C 180,E1 -16399.244,E2 -16399.244} C_VEL
LIN {X 0,Y 298.45,Z 293.121,A -85,B 0,C 180,E1 -16403.598,E2 -16403.598} C_VEL
LIN {X 0,Y 298.483,Z 293.115,A -85,B 0,C 180,E1 -16406.575,E2 -16406.575} C_VEL
LIN {X 0,Y 298.414,Z 293.125,A -85,B 0,C 180,E1 -16409.642,E2 -16409.642} C_VEL
LIN {X 0,Y 298.389,Z 293.129,A -85,B 0,C 180,E1 -16412.801,E2 -16412.801} C_VEL
LIN {X 0,Y 298.475,Z 293.119,A -85,B 0,C 180,E1 -16417.056,E2 -16417.056} C_VEL
LIN {X 0,Y 300.039,Z 300.615,A -85,B 0,C 180,E1 -16419.882,E2 -16419.882} C_VEL
LIN {X 0,Y 304.439,Z 312.103,A -85,B 0,C 180,E1 -16420.597,E2 -16420.597} C_VEL
LIN {X 0,Y 307.632,Z 328.348,A -85,B 0,C 180,E1 -16421.303,E2 -16421.303} C_VEL
LIN {X 0,Y 306.311,Z 377.675,A -85,B 0,C 180,E1 -16422.542,E2 -16422.542} C_VEL
LIN {X 0,Y 305.789,Z 387.484,A -85,B 0,C 180,E1 -16422.962,E2 -16422.962} C_VEL
LIN {X 0,Y 305.054,Z 399.079,A -85,B 0,C 180,E1 -16423.722,E2 -16423.722} C_VEL
LIN {X 0,Y 303.988,Z 409.467,A -85,B 0,C 180,E1 -16424.692,E2 -16424.692} C_VEL
LIN {X 0,Y 303.02,Z 417.717,A -85,B 0,C 180,E1 -16425.679,E2 -16425.679} C_VEL
LIN {X 0,Y 301.9,Z 425.692,A -85,B 0,C 180,E1 -16426.858,E2 -16426.858} C_VEL
LIN {X 0,Y 300.928,Z 432.027,A -85,B 0,C 180,E1 -16427.999,E2 -16427.999} C_VEL
LIN {X 0,Y 299.894,Z 438.596,A -85,B 0,C 180,E1 -16429.436,E2 -16429.436} C_VEL
LIN {X 0,Y 298.903,Z 445.051,A -85,B 0,C 180,E1 -16431.194,E2 -16431.194} C_VEL
LIN {X 0,Y 297.938,Z 450.91,A -85,B 0,C 180,E1 -16433.324,E2 -16433.324} C_VEL
LIN {X 0,Y 297.39,Z 453.735,A -85,B 0,C 180,E1 -16434.622,E2 -16434.622} C_VEL
LIN {X 0,Y 297.119,Z 455.852,A -85,B 0,C 180,E1 -16435.882,E2 -16435.882} C_VEL
LIN {X 0,Y 296.859,Z 457.317,A -85,B 0,C 180,E1 -16437.01,E2 -16437.01} C_VEL
LIN {X 0,Y 296.585,Z 458.815,A -85,B 0,C 180,E1 -16438.58,E2 -16438.58} C_VEL
LIN {X 0,Y 296.35,Z 459.634,A -85,B 0,C 180,E1 -16440.132,E2 -16440.132} C_VEL
LIN {X 0,Y 296.259,Z 459.808,A -85,B 0,C 180,E1 -16441.678,E2 -16441.678} C_VEL
LIN {X 0,Y 296.274,Z 459.349,A -85,B 0,C 180,E1 -16443.212,E2 -16443.212} C_VEL
LIN {X 0,Y 296.394,Z 458.231,A -85,B 0,C 180,E1 -16444.736,E2 -16444.736} C_VEL
LIN {X 0,Y 296.645,Z 456.436,A -85,B 0,C 180,E1 -16446.25,E2 -16446.25} C_VEL
LIN {X 0,Y 297.072,Z 452.514,A -85,B 0,C 180,E1 -16448.489,E2 -16448.489} C_VEL
LIN {X 0,Y 297.538,Z 447.994,A -85,B 0,C 180,E1 -16450.331,E2 -16450.331} C_VEL
LIN {X 0,Y 298.034,Z 443.402,A -85,B 0,C 180,E1 -16451.815,E2 -16451.815} C_VEL
LIN {X 0,Y 298.7,Z 437.957,A -85,B 0,C 180,E1 -16453.249,E2 -16453.249} C_VEL
LIN {X 0,Y 299.267,Z 433.081,A -85,B 0,C 180,E1 -16454.334,E2 -16454.334} C_VEL
LIN {X 0,Y 300.025,Z 426.321,A -85,B 0,C 180,E1 -16455.589,E2 -16455.589} C_VEL
LIN {X 0,Y 300.796,Z 419.356,A -85,B 0,C 180,E1 -16456.661,E2 -16456.661} C_VEL
LIN {X 0,Y 301.658,Z 410.828,A -85,B 0,C 180,E1 -16457.726,E2 -16457.726} C_VEL
LIN {X 0,Y 302.386,Z 401.963,A -85,B 0,C 180,E1 -16458.606,E2 -16458.606} C_VEL
LIN {X 0,Y 302.914,Z 392.92,A -85,B 0,C 180,E1 -16459.304,E2 -16459.304} C_VEL
LIN {X 0,Y 303.51,Z 381.831,A -85,B 0,C 180,E1 -16459.915,E2 -16459.915} C_VEL
LIN {X 0,Y 303.957,Z 367.458,A -85,B 0,C 180,E1 -16460.35,E2 -16460.35} C_VEL
LIN {X 0,Y 304.632,Z 326.347,A -85,B 0,C 180,E1 -16461.355,E2 -16461.355} C_VEL
LIN {X 0,Y 300.161,Z 302.16,A -85,B 0,C 180,E1 -16462.242,E2 -16462.242} C_VEL
LIN {X 0,Y 299.82,Z 300.595,A -85,B 0,C 180,E1 -16462.339,E2 -16462.339} C_VEL
LIN {X 0,Y 298.934,Z 294.594,A -85,B 0,C 180,E1 -16464.604,E2 -16464.604} C_VEL
LIN {X 0,Y 298.649,Z 293.098,A -85,B 0,C 180,E1 -16465.276,E2 -16465.276} C_VEL
LIN {X 0,Y 298.924,Z 293.061,A -85,B 0,C 180,E1 -16468.653,E2 -16468.653} C_VEL
LIN {X 0,Y 298.924,Z 293.061,A -85,B 0,C 180,E1 -16471.347,E2 -16471.347} C_VEL
LIN {X 0,Y 298.646,Z 293.093,A -85,B 0,C 180,E1 -16475.401,E2 -16475.401} C_VEL
LIN {X 0,Y 298.715,Z 293.09,A -85,B 0,C 180,E1 -16478.115,E2 -16478.115} C_VEL
LIN {X 0,Y 298.555,Z 293.108,A -85,B 0,C 180,E1 -16482.231,E2 -16482.231} C_VEL
LIN {X 0,Y 298.549,Z 293.106,A -85,B 0,C 180,E1 -16485.168,E2 -16485.168} C_VEL
LIN {X 0,Y 298.504,Z 293.11,A -85,B 0,C 180,E1 -16489.245,E2 -16489.245} C_VEL
LIN {X 0,Y 298.429,Z 293.119,A -85,B 0,C 180,E1 -16493.599,E2 -16493.599} C_VEL
LIN {X 0,Y 298.485,Z 293.117,A -85,B 0,C 180,E1 -16496.574,E2 -16496.574} C_VEL
LIN {X 0,Y 298.42,Z 293.123,A -85,B 0,C 180,E1 -16499.64,E2 -16499.64} C_VEL
LIN {X 0,Y 298.394,Z 293.127,A -85,B 0,C 180,E1 -16502.799,E2 -16502.799} C_VEL
LIN {X 0,Y 298.442,Z 293.121,A -85,B 0,C 180,E1 -16506.806,E2 -16506.806} C_VEL
LIN {X 0,Y 298.385,Z 293.128,A -85,B 0,C 180,E1 -16511.087,E2 -16511.087} C_VEL
LIN {X 0,Y 298.413,Z 293.122,A -85,B 0,C 180,E1 -16514.952,E2 -16514.952} C_VEL
LIN {X 0,Y 298.447,Z 293.118,A -85,B 0,C 180,E1 -16518.749,E2 -16518.749} C_VEL
LIN {X 0,Y 298.46,Z 293.115,A -85,B 0,C 180,E1 -16523.187,E2 -16523.187} C_VEL
LIN {X 0,Y 298.39,Z 293.124,A -85,B 0,C 180,E1 -16527.199,E2 -16527.199} C_VEL
LIN {X 0,Y 298.444,Z 293.121,A -85,B 0,C 180,E1 -16531.737,E2 -16531.737} C_VEL
LIN {X 0,Y 298.478,Z 293.114,A -85,B 0,C 180,E1 -16534.923,E2 -16534.923} C_VEL
LIN {X 0,Y 298.412,Z 293.12,A -85,B 0,C 180,E1 -16537.57,E2 -16537.57} C_VEL
LIN {X 0,Y 297.776,Z 293.203,A -85,B 0,C 180,E1 -16538.697,E2 -16538.697} C_VEL
LIN {X 0,Y 294.965,Z 293.554,A -85,B 0,C 180,E1 -16540.533,E2 -16540.533} C_VEL
LIN {X 0,Y 292.573,Z 293.85,A -85,B 0,C 180,E1 -16542.023,E2 -16542.023} C_VEL
LIN {X 0,Y 291.553,Z 293.977,A -85,B 0,C 180,E1 -16543.176,E2 -16543.176} C_VEL
LIN {X 0,Y 291.475,Z 293.985,A -85,B 0,C 180,E1 -16543.567,E2 -16543.567} C_VEL
LIN {X 0,Y 291.511,Z 293.982,A -85,B 0,C 180,E1 -16547.468,E2 -16547.468} C_VEL
LIN {X 0,Y 291.679,Z 293.959,A -85,B 0,C 180,E1 -16551.687,E2 -16551.687} C_VEL
LIN {X 0,Y 291.617,Z 293.966,A -85,B 0,C 180,E1 -16554.468,E2 -16554.468} C_VEL
LIN {X 0,Y 291.88,Z 293.936,A -85,B 0,C 180,E1 -16558.62,E2 -16558.62} C_VEL
LIN {X 0,Y 291.881,Z 293.94,A -85,B 0,C 180,E1 -16561.38,E2 -16561.38} C_VEL
LIN {X 0,Y 291.726,Z 293.956,A -85,B 0,C 180,E1 -16566.918,E2 -16566.918} C_VEL
LIN {X 0,Y 291.568,Z 293.975,A -85,B 0,C 180,E1 -16569.714,E2 -16569.714} C_VEL
LIN {X 0,Y 291.514,Z 293.984,A -85,B 0,C 180,E1 -16573.95,E2 -16573.95} C_VEL
LIN {X 0,Y 291.477,Z 293.986,A -85,B 0,C 180,E1 -16576.818,E2 -16576.818} C_VEL
LIN {X 0,Y 291.443,Z 293.993,A -85,B 0,C 180,E1 -16579.875,E2 -16579.875} C_VEL
LIN {X 0,Y 291.375,Z 294.002,A -85,B 0,C 180,E1 -16584.207,E2 -16584.207} C_VEL
LIN {X 0,Y 291.412,Z 293.995,A -85,B 0,C 180,E1 -16587.272,E2 -16587.272} C_VEL
LIN {X 0,Y 291.326,Z 294.007,A -85,B 0,C 180,E1 -16590.438,E2 -16590.438} C_VEL
LIN {X 0,Y 291.338,Z 294.005,A -85,B 0,C 180,E1 -16593.699,E2 -16593.699} C_VEL
LIN {X 0,Y 291.369,Z 293.999,A -85,B 0,C 180,E1 -16597.254,E2 -16597.254} C_VEL
LIN {X 0,Y 291.327,Z 294.004,A -85,B 0,C 180,E1 -16600.643,E2 -16600.643} C_VEL
LIN {X 0,Y 291.309,Z 294.009,A -85,B 0,C 180,E1 -16604.398,E2 -16604.398} C_VEL
LIN {X 0,Y 291.322,Z 294.008,A -85,B 0,C 180,E1 -16608.405,E2 -16608.405} C_VEL
LIN {X 0,Y 291.343,Z 294.007,A -85,B 0,C 180,E1 -16611.158,E2 -16611.158} C_VEL
LIN {X 0,Y 291.357,Z 294.004,A -85,B 0,C 180,E1 -16614.627,E2 -16614.627} C_VEL
LIN {X 0,Y 291.363,Z 294.002,A -85,B 0,C 180,E1 -16617.951,E2 -16617.951} C_VEL
LIN {X 0,Y 291.467,Z 294.152,A -85,B 0,C 180,E1 -16621.562,E2 -16621.562} C_VEL
LIN {X 0,Y 293.47,Z 304.948,A -85,B 0,C 180,E1 -16625.508,E2 -16625.508} C_VEL
LIN {X 0,Y 293.71,Z 308.497,A -85,B 0,C 180,E1 -16626.746,E2 -16626.746} C_VEL
LIN {X 0,Y 292.786,Z 316.078,A -85,B 0,C 180,E1 -16629.275,E2 -16629.275} C_VEL
LIN {X 0,Y 297.473,Z 351.565,A -85,B 0,C 180,E1 -16630.511,E2 -16630.511} C_VEL
LIN {X 0,Y 296.706,Z 393.443,A -85,B 0,C 180,E1 -16631.597,E2 -16631.597} C_VEL
LIN {X 0,Y 296.16,Z 403.401,A -85,B 0,C 180,E1 -16632.032,E2 -16632.032} C_VEL
LIN {X 0,Y 295.419,Z 413.712,A -85,B 0,C 180,E1 -16632.701,E2 -16632.701} C_VEL
LIN {X 0,Y 294.439,Z 424.633,A -85,B 0,C 180,E1 -16633.713,E2 -16633.713} C_VEL
LIN {X 0,Y 293.569,Z 433.089,A -85,B 0,C 180,E1 -16634.732,E2 -16634.732} C_VEL
LIN {X 0,Y 292.672,Z 441.076,A -85,B 0,C 180,E1 -16635.929,E2 -16635.929} C_VEL
LIN {X 0,Y 291.919,Z 447.678,A -85,B 0,C 180,E1 -16637.133,E2 -16637.133} C_VEL
LIN {X 0,Y 291.169,Z 453.95,A -85,B 0,C 180,E1 -16638.514,E2 -16638.514} C_VEL
LIN {X 0,Y 290.566,Z 459.151,A -85,B 0,C 180,E1 -16639.901,E2 -16639.901} C_VEL
LIN {X 0,Y 290.231,Z 462.512,A -85,B 0,C 180,E1 -16640.944,E2 -16640.944} C_VEL
LIN {X 0,Y 289.852,Z 466.291,A -85,B 0,C 180,E1 -16642.337,E2 -16642.337} C_VEL
LIN {X 0,Y 289.535,Z 470.577,A -85,B 0,C 180,E1 -16644.428,E2 -16644.428} C_VEL
LIN {X 0,Y 289.465,Z 472.754,A -85,B 0,C 180,E1 -16645.823,E2 -16645.823} C_VEL
LIN {X 0,Y 289.471,Z 474.366,A -85,B 0,C 180,E1 -16647.217,E2 -16647.217} C_VEL
LIN {X 0,Y 289.408,Z 475.363,A -85,B 0,C 180,E1 -16648.609,E2 -16648.609} C_VEL
LIN {X 0,Y 289.434,Z 475.867,A -85,B 0,C 180,E1 -16650,E2 -16650} C_VEL
LIN {X 0,Y 289.407,Z 475.899,A -85,B 0,C 180,E1 -16651.391,E2 -16651.391} C_VEL
LIN {X 0,Y 289.448,Z 475.465,A -85,B 0,C 180,E1 -16652.783,E2 -16652.783} C_VEL
LIN {X 0,Y 289.466,Z 474.466,A -85,B 0,C 180,E1 -16654.177,E2 -16654.177} C_VEL
LIN {X 0,Y 289.55,Z 472.817,A -85,B 0,C 180,E1 -16655.642,E2 -16655.642} C_VEL
LIN {X 0,Y 289.925,Z 469.652,A -85,B 0,C 180,E1 -16657.661,E2 -16657.661} C_VEL
LIN {X 0,Y 290.586,Z 464.965,A -85,B 0,C 180,E1 -16659.747,E2 -16659.747} C_VEL
LIN {X 0,Y 291.371,Z 459.851,A -85,B 0,C 180,E1 -16661.478,E2 -16661.478} C_VEL
LIN {X 0,Y 292.244,Z 454.882,A -85,B 0,C 180,E1 -16662.852,E2 -16662.852} C_VEL
LIN {X 0,Y 293.194,Z 448.906,A -85,B 0,C 180,E1 -16664.223,E2 -16664.223} C_VEL
LIN {X 0,Y 294.307,Z 441.649,A -85,B 0,C 180,E1 -16665.583,E2 -16665.583} C_VEL
LIN {X 0,Y 295.499,Z 433.912,A -85,B 0,C 180,E1 -16666.76,E2 -16666.76} C_VEL
LIN {X 0,Y 296.649,Z 425.789,A -85,B 0,C 180,E1 -16667.759,E2 -16667.759} C_VEL
LIN {X 0,Y 297.535,Z 417.388,A -85,B 0,C 180,E1 -16668.595,E2 -16668.595} C_VEL
LIN {X 0,Y 298.517,Z 407.447,A -85,B 0,C 180,E1 -16669.346,E2 -16669.346} C_VEL
LIN {X 0,Y 299.483,Z 395.007,A -85,B 0,C 180,E1 -16669.967,E2 -16669.967} C_VEL
LIN {X 0,Y 300.126,Z 374.751,A -85,B 0,C 180,E1 -16670.523,E2 -16670.523} C_VEL
LIN {X 0,Y 300.494,Z 352.143,A -85,B 0,C 180,E1 -16671.105,E2 -16671.105} C_VEL
LIN {X 0,Y 297.526,Z 331.94,A -85,B 0,C 180,E1 -16671.919,E2 -16671.919} C_VEL
LIN {X 0,Y 294.103,Z 314.903,A -85,B 0,C 180,E1 -16672.756,E2 -16672.756} C_VEL
LIN {X 0,Y 294.579,Z 311.317,A -85,B 0,C 180,E1 -16673.927,E2 -16673.927} C_VEL
LIN {X 0,Y 293.865,Z 305.808,A -85,B 0,C 180,E1 -16675.877,E2 -16675.877} C_VEL
LIN {X 0,Y 291.982,Z 296.726,A -85,B 0,C 180,E1 -16679.283,E2 -16679.283} C_VEL
LIN {X 0,Y 291.37,Z 294.006,A -85,B 0,C 180,E1 -16680.432,E2 -16680.432} C_VEL
LIN {X 0,Y 291.366,Z 294.004,A -85,B 0,C 180,E1 -16684.905,E2 -16684.905} C_VEL
LIN {X 0,Y 291.372,Z 294.006,A -85,B 0,C 180,E1 -16687.253,E2 -16687.253} C_VEL
LIN {X 0,Y 291.328,Z 294.016,A -85,B 0,C 180,E1 -16690.642,E2 -16690.642} C_VEL
LIN {X 0,Y 291.285,Z 294.018,A -85,B 0,C 180,E1 -16694.401,E2 -16694.401} C_VEL
LIN {X 0,Y 291.32,Z 294.006,A -85,B 0,C 180,E1 -16698.404,E2 -16698.404} C_VEL
LIN {X 0,Y 291.347,Z 294.008,A -85,B 0,C 180,E1 -16701.158,E2 -16701.158} C_VEL
LIN {X 0,Y 291.355,Z 294.003,A -85,B 0,C 180,E1 -16704.625,E2 -16704.625} C_VEL
LIN {X 0,Y 291.364,Z 293.995,A -85,B 0,C 180,E1 -16707.95,E2 -16707.95} C_VEL
LIN {X 0,Y 291.375,Z 293.999,A -85,B 0,C 180,E1 -16711.158,E2 -16711.158} C_VEL
LIN {X 0,Y 291.406,Z 293.995,A -85,B 0,C 180,E1 -16714.271,E2 -16714.271} C_VEL
LIN {X 0,Y 291.365,Z 293.995,A -85,B 0,C 180,E1 -16717.298,E2 -16717.298} C_VEL
LIN {X 0,Y 291.45,Z 293.99,A -85,B 0,C 180,E1 -16720.27,E2 -16720.27} C_VEL
LIN {X 0,Y 291.532,Z 293.968,A -85,B 0,C 180,E1 -16724.634,E2 -16724.634} C_VEL
LIN {X 0,Y 291.526,Z 293.977,A -85,B 0,C 180,E1 -16728.88,E2 -16728.88} C_VEL
LIN {X 0,Y 291.679,Z 293.953,A -85,B 0,C 180,E1 -16731.688,E2 -16731.688} C_VEL
LIN {X 0,Y 291.616,Z 293.971,A -85,B 0,C 180,E1 -16734.468,E2 -16734.468} C_VEL
LIN {X 0,Y 291.879,Z 293.933,A -85,B 0,C 180,E1 -16738.62,E2 -16738.62} C_VEL
LIN {X 0,Y 291.879,Z 293.928,A -85,B 0,C 180,E1 -16741.38,E2 -16741.38} C_VEL
LIN {X 0,Y 291.643,Z 293.961,A -85,B 0,C 180,E1 -16746.536,E2 -16746.536} C_VEL
LIN {X 0,Y 291.563,Z 293.98,A -85,B 0,C 180,E1 -16749.714,E2 -16749.714} C_VEL
LIN {X 0,Y 291.513,Z 293.987,A -85,B 0,C 180,E1 -16753.951,E2 -16753.951} C_VEL
LIN {X 0,Y 291.478,Z 293.983,A -85,B 0,C 180,E1 -16756.819,E2 -16756.819} C_VEL
LIN {X 0,Y 291.444,Z 293.992,A -85,B 0,C 180,E1 -16759.876,E2 -16759.876} C_VEL
LIN {X 0,Y 291.393,Z 294.001,A -85,B 0,C 180,E1 -16764.206,E2 -16764.206} C_VEL
LIN {X 0,Y 291.416,Z 293.996,A -85,B 0,C 180,E1 -16767.272,E2 -16767.272} C_VEL
LIN {X 0,Y 291.331,Z 294.008,A -85,B 0,C 180,E1 -16770.438,E2 -16770.438} C_VEL
LIN {X 0,Y 291.339,Z 294.01,A -85,B 0,C 180,E1 -16773.699,E2 -16773.699} C_VEL
LIN {X 0,Y 291.435,Z 294.196,A -85,B 0,C 180,E1 -16776.645,E2 -16776.645} C_VEL
LIN {X 0,Y 292.93,Z 301.095,A -85,B 0,C 180,E1 -16779.229,E2 -16779.229} C_VEL
LIN {X 0,Y 298.266,Z 314.49,A -85,B 0,C 180,E1 -16780.113,E2 -16780.113} C_VEL
LIN {X 0,Y 301.137,Z 329.364,A -85,B 0,C 180,E1 -16780.776,E2 -16780.776} C_VEL
LIN {X 0,Y 299.78,Z 377.972,A -85,B 0,C 180,E1 -16782.026,E2 -16782.026} C_VEL
LIN {X 0,Y 299.181,Z 388.529,A -85,B 0,C 180,E1 -16782.493,E2 -16782.493} C_VEL
LIN {X 0,Y 298.325,Z 400.546,A -85,B 0,C 180,E1 -16783.337,E2 -16783.337} C_VEL
LIN {X 0,Y 297.41,Z 408.931,A -85,B 0,C 180,E1 -16784.13,E2 -16784.13} C_VEL
LIN {X 0,Y 296.432,Z 417.238,A -85,B 0,C 180,E1 -16785.13,E2 -16785.13} C_VEL
LIN {X 0,Y 295.229,Z 425.395,A -85,B 0,C 180,E1 -16786.344,E2 -16786.344} C_VEL
LIN {X 0,Y 294.191,Z 432.023,A -85,B 0,C 180,E1 -16787.554,E2 -16787.554} C_VEL
LIN {X 0,Y 293.227,Z 437.589,A -85,B 0,C 180,E1 -16788.769,E2 -16788.769} C_VEL
LIN {X 0,Y 292.279,Z 443.365,A -85,B 0,C 180,E1 -16790.305,E2 -16790.305} C_VEL
LIN {X 0,Y 291.366,Z 448.615,A -85,B 0,C 180,E1 -16792.044,E2 -16792.044} C_VEL
LIN {X 0,Y 290.711,Z 452.491,A -85,B 0,C 180,E1 -16793.681,E2 -16793.681} C_VEL
LIN {X 0,Y 290.115,Z 455.702,A -85,B 0,C 180,E1 -16795.452,E2 -16795.452} C_VEL
LIN {X 0,Y 289.638,Z 458.53,A -85,B 0,C 180,E1 -16797.737,E2 -16797.737} C_VEL
LIN {X 0,Y 289.352,Z 459.624,A -85,B 0,C 180,E1 -16799.333,E2 -16799.333} C_VEL
LIN {X 0,Y 289.189,Z 460.052,A -85,B 0,C 180,E1 -16801.032,E2 -16801.032} C_VEL
LIN {X 0,Y 289.145,Z 459.787,A -85,B 0,C 180,E1 -16802.497,E2 -16802.497} C_VEL
LIN {X 0,Y 289.253,Z 458.916,A -85,B 0,C 180,E1 -16804.066,E2 -16804.066} C_VEL
LIN {X 0,Y 289.587,Z 456.498,A -85,B 0,C 180,E1 -16806.395,E2 -16806.395} C_VEL
LIN {X 0,Y 290.014,Z 452.474,A -85,B 0,C 180,E1 -16808.685,E2 -16808.685} C_VEL
LIN {X 0,Y 290.539,Z 447.73,A -85,B 0,C 180,E1 -16810.63,E2 -16810.63} C_VEL
LIN {X 0,Y 291.189,Z 442.031,A -85,B 0,C 180,E1 -16812.441,E2 -16812.441} C_VEL
LIN {X 0,Y 292.19,Z 434.153,A -85,B 0,C 180,E1 -16814.385,E2 -16814.385} C_VEL
LIN {X 0,Y 293.149,Z 425.874,A -85,B 0,C 180,E1 -16815.952,E2 -16815.952} C_VEL
LIN {X 0,Y 293.934,Z 418.792,A -85,B 0,C 180,E1 -16817.047,E2 -16817.047} C_VEL
LIN {X 0,Y 294.809,Z 410.43,A -85,B 0,C 180,E1 -16818.098,E2 -16818.098} C_VEL
LIN {X 0,Y 295.486,Z 402.708,A -85,B 0,C 180,E1 -16818.881,E2 -16818.881} C_VEL
LIN {X 0,Y 296.006,Z 394.165,A -85,B 0,C 180,E1 -16819.57,E2 -16819.57} C_VEL
LIN {X 0,Y 296.519,Z 384.432,A -85,B 0,C 180,E1 -16820.149,E2 -16820.149} C_VEL
LIN {X 0,Y 297,Z 372.567,A -85,B 0,C 180,E1 -16820.595,E2 -16820.595} C_VEL
LIN {X 0,Y 297.807,Z 327.044,A -85,B 0,C 180,E1 -16821.732,E2 -16821.732} C_VEL
LIN {X 0,Y 293.642,Z 304.339,A -85,B 0,C 180,E1 -16822.587,E2 -16822.587} C_VEL
LIN {X 0,Y 292.73,Z 300.809,A -85,B 0,C 180,E1 -16822.759,E2 -16822.759} C_VEL
LIN {X 0,Y 292.081,Z 296.367,A -85,B 0,C 180,E1 -16824.477,E2 -16824.477} C_VEL
LIN {X 0,Y 291.599,Z 293.977,A -85,B 0,C 180,E1 -16825.508,E2 -16825.508} C_VEL
LIN {X 0,Y 291.89,Z 293.937,A -85,B 0,C 180,E1 -16828.62,E2 -16828.62} C_VEL
LIN {X 0,Y 291.89,Z 293.937,A -85,B 0,C 180,E1 -16831.38,E2 -16831.38} C_VEL
LIN {X 0,Y 291.615,Z 293.97,A -85,B 0,C 180,E1 -16835.532,E2 -16835.532} C_VEL
LIN {X 0,Y 291.676,Z 293.963,A -85,B 0,C 180,E1 -16838.919,E2 -16838.919} C_VEL
LIN {X 0,Y 291.52,Z 293.983,A -85,B 0,C 180,E1 -16842.531,E2 -16842.531} C_VEL
LIN {X 0,Y 291.508,Z 293.983,A -85,B 0,C 180,E1 -16845.378,E2 -16845.378} C_VEL
LIN {X 0,Y 291.424,Z 293.991,A -85,B 0,C 180,E1 -16849.859,E2 -16849.859} C_VEL
LIN {X 0,Y 291.382,Z 293.997,A -85,B 0,C 180,E1 -16854.206,E2 -16854.206} C_VEL
LIN {X 0,Y 291.42,Z 293.997,A -85,B 0,C 180,E1 -16857.271,E2 -16857.271} C_VEL
LIN {X 0,Y 291.336,Z 294.006,A -85,B 0,C 180,E1 -16860.436,E2 -16860.436} C_VEL
LIN {X 0,Y 291.343,Z 294.003,A -85,B 0,C 180,E1 -16863.697,E2 -16863.697} C_VEL
LIN {X 0,Y 291.37,Z 294.006,A -85,B 0,C 180,E1 -16867.252,E2 -16867.252} C_VEL
LIN {X 0,Y 291.33,Z 294.004,A -85,B 0,C 180,E1 -16870.641,E2 -16870.641} C_VEL
LIN {X 0,Y 291.339,Z 294.002,A -85,B 0,C 180,E1 -16874.391,E2 -16874.391} C_VEL
LIN {X 0,Y 291.382,Z 293.999,A -85,B 0,C 180,E1 -16878.39,E2 -16878.39} C_VEL
LIN {X 0,Y 291.374,Z 294,A -85,B 0,C 180,E1 -16881.161,E2 -16881.161} C_VEL
LIN {X 0,Y 291.38,Z 293.994,A -85,B 0,C 180,E1 -16884.628,E2 -16884.628} C_VEL
LIN {X 0,Y 291.366,Z 294.003,A -85,B 0,C 180,E1 -16887.95,E2 -16887.95} C_VEL
LIN {X 0,Y 291.375,Z 293.999,A -85,B 0,C 180,E1 -16891.157,E2 -16891.157} C_VEL
LIN {X 0,Y 291.41,Z 293.998,A -85,B 0,C 180,E1 -16894.271,E2 -16894.271} C_VEL
LIN {X 0,Y 291.359,Z 293.996,A -85,B 0,C 180,E1 -16897.557,E2 -16897.557} C_VEL
LIN {X 0,Y 291.451,Z 293.988,A -85,B 0,C 180,E1 -16900.269,E2 -16900.269} C_VEL
LIN {X 0,Y 291.475,Z 293.985,A -85,B 0,C 180,E1 -16903.567,E2 -16903.567} C_VEL
LIN {X 0,Y 290.813,Z 294.073,A -85,B 0,C 180,E1 -16904.72,E2 -16904.72} C_VEL
LIN {X 0,Y 287.952,Z 294.431,A -85,B 0,C 180,E1 -16906.599,E2 -16906.599} C_VEL
LIN {X 0,Y 285.545,Z 294.727,A -85,B 0,C 180,E1 -16908.124,E2 -16908.124} C_VEL
LIN {X 0,Y 284.548,Z 294.85,A -85,B 0,C 180,E1 -16909.306,E2 -16909.306} C_VEL
LIN {X 0,Y 284.487,Z 294.856,A -85,B 0,C 180,E1 -16909.706,E2 -16909.706} C_VEL
LIN {X 0,Y 284.677,Z 294.833,A -85,B 0,C 180,E1 -16912.909,E2 -16912.909} C_VEL
LIN {X 0,Y 284.846,Z 294.811,A -85,B 0,C 180,E1 -16918.586,E2 -16918.586} C_VEL
LIN {X 0,Y 284.847,Z 294.816,A -85,B 0,C 180,E1 -16921.414,E2 -16921.414} C_VEL
LIN {X 0,Y 284.677,Z 294.835,A -85,B 0,C 180,E1 -16927.09,E2 -16927.09} C_VEL
LIN {X 0,Y 284.512,Z 294.851,A -85,B 0,C 180,E1 -16929.957,E2 -16929.957} C_VEL
LIN {X 0,Y 284.47,Z 294.86,A -85,B 0,C 180,E1 -16934.303,E2 -16934.303} C_VEL
LIN {X 0,Y 284.414,Z 294.868,A -85,B 0,C 180,E1 -16937.249,E2 -16937.249} C_VEL
LIN {X 0,Y 284.37,Z 294.87,A -85,B 0,C 180,E1 -16940.243,E2 -16940.243} C_VEL
LIN {X 0,Y 284.33,Z 294.877,A -85,B 0,C 180,E1 -16944.847,E2 -16944.847} C_VEL
LIN {X 0,Y 284.321,Z 294.883,A -85,B 0,C 180,E1 -16948.012,E2 -16948.012} C_VEL
LIN {X 0,Y 284.286,Z 294.881,A -85,B 0,C 180,E1 -16951.275,E2 -16951.275} C_VEL
LIN {X 0,Y 284.335,Z 294.877,A -85,B 0,C 180,E1 -16955.349,E2 -16955.349} C_VEL
LIN {X 0,Y 284.306,Z 294.882,A -85,B 0,C 180,E1 -16958.17,E2 -16958.17} C_VEL
LIN {X 0,Y 284.264,Z 294.882,A -85,B 0,C 180,E1 -16962.125,E2 -16962.125} C_VEL
LIN {X 0,Y 284.264,Z 294.886,A -85,B 0,C 180,E1 -16966.193,E2 -16966.193} C_VEL
LIN {X 0,Y 284.302,Z 294.881,A -85,B 0,C 180,E1 -16970.025,E2 -16970.025} C_VEL
LIN {X 0,Y 284.327,Z 294.879,A -85,B 0,C 180,E1 -16973.615,E2 -16973.615} C_VEL
LIN {X 0,Y 284.303,Z 294.885,A -85,B 0,C 180,E1 -16977.191,E2 -16977.191} C_VEL
LIN {X 0,Y 284.389,Z 295.061,A -85,B 0,C 180,E1 -16981.293,E2 -16981.293} C_VEL
LIN {X 0,Y 286.427,Z 305.869,A -85,B 0,C 180,E1 -16985.348,E2 -16985.348} C_VEL
LIN {X 0,Y 286.717,Z 309.156,A -85,B 0,C 180,E1 -16986.528,E2 -16986.528} C_VEL
LIN {X 0,Y 285.893,Z 316,A -85,B 0,C 180,E1 -16988.855,E2 -16988.855} C_VEL
LIN {X 0,Y 290.722,Z 352.86,A -85,B 0,C 180,E1 -16990.152,E2 -16990.152} C_VEL
LIN {X 0,Y 289.885,Z 393.273,A -85,B 0,C 180,E1 -16991.223,E2 -16991.223} C_VEL
LIN {X 0,Y 289.294,Z 403.507,A -85,B 0,C 180,E1 -16991.682,E2 -16991.682} C_VEL
LIN {X 0,Y 288.547,Z 413.729,A -85,B 0,C 180,E1 -16992.367,E2 -16992.367} C_VEL
LIN {X 0,Y 287.609,Z 423.825,A -85,B 0,C 180,E1 -16993.315,E2 -16993.315} C_VEL
LIN {X 0,Y 286.711,Z 432.391,A -85,B 0,C 180,E1 -16994.358,E2 -16994.358} C_VEL
LIN {X 0,Y 285.788,Z 440.465,A -85,B 0,C 180,E1 -16995.583,E2 -16995.583} C_VEL
LIN {X 0,Y 284.979,Z 447.134,A -85,B 0,C 180,E1 -16996.814,E2 -16996.814} C_VEL
LIN {X 0,Y 284.198,Z 453.465,A -85,B 0,C 180,E1 -16998.228,E2 -16998.228} C_VEL
LIN {X 0,Y 283.532,Z 458.715,A -85,B 0,C 180,E1 -16999.648,E2 -16999.648} C_VEL
LIN {X 0,Y 283.192,Z 462.122,A -85,B 0,C 180,E1 -17000.717,E2 -17000.717} C_VEL
LIN {X 0,Y 282.789,Z 465.931,A -85,B 0,C 180,E1 -17002.144,E2 -17002.144} C_VEL
LIN {X 0,Y 282.481,Z 470.266,A -85,B 0,C 180,E1 -17004.289,E2 -17004.289} C_VEL
LIN {X 0,Y 282.37,Z 472.477,A -85,B 0,C 180,E1 -17005.718,E2 -17005.718} C_VEL
LIN {X 0,Y 282.377,Z 474.099,A -85,B 0,C 180,E1 -17007.147,E2 -17007.147} C_VEL
LIN {X 0,Y 282.333,Z 475.119,A -85,B 0,C 180,E1 -17008.574,E2 -17008.574} C_VEL
LIN {X 0,Y 282.353,Z 475.654,A -85,B 0,C 180,E1 -17010,E2 -17010} C_VEL
LIN {X 0,Y 282.331,Z 475.718,A -85,B 0,C 180,E1 -17011.426,E2 -17011.426} C_VEL
LIN {X 0,Y 282.356,Z 475.308,A -85,B 0,C 180,E1 -17012.853,E2 -17012.853} C_VEL
LIN {X 0,Y 282.373,Z 474.314,A -85,B 0,C 180,E1 -17014.282,E2 -17014.282} C_VEL
LIN {X 0,Y 282.577,Z 471.906,A -85,B 0,C 180,E1 -17016.426,E2 -17016.426} C_VEL
LIN {X 0,Y 283.077,Z 468.161,A -85,B 0,C 180,E1 -17018.567,E2 -17018.567} C_VEL
LIN {X 0,Y 283.595,Z 464.971,A -85,B 0,C 180,E1 -17019.989,E2 -17019.989} C_VEL
LIN {X 0,Y 284.425,Z 459.911,A -85,B 0,C 180,E1 -17021.762,E2 -17021.762} C_VEL
LIN {X 0,Y 285.333,Z 454.994,A -85,B 0,C 180,E1 -17023.169,E2 -17023.169} C_VEL
LIN {X 0,Y 286.319,Z 449.079,A -85,B 0,C 180,E1 -17024.572,E2 -17024.572} C_VEL
LIN {X 0,Y 287.503,Z 441.894,A -85,B 0,C 180,E1 -17025.962,E2 -17025.962} C_VEL
LIN {X 0,Y 288.733,Z 434.245,A -85,B 0,C 180,E1 -17027.165,E2 -17027.165} C_VEL
LIN {X 0,Y 289.932,Z 426.237,A -85,B 0,C 180,E1 -17028.185,E2 -17028.185} C_VEL
LIN {X 0,Y 290.849,Z 417.994,A -85,B 0,C 180,E1 -17029.038,E2 -17029.038} C_VEL
LIN {X 0,Y 291.721,Z 409.647,A -85,B 0,C 180,E1 -17029.711,E2 -17029.711} C_VEL
LIN {X 0,Y 292.589,Z 400.432,A -85,B 0,C 180,E1 -17030.256,E2 -17030.256} C_VEL
LIN {X 0,Y 293.172,Z 390.228,A -85,B 0,C 180,E1 -17030.665,E2 -17030.665} C_VEL
LIN {X 0,Y 293.994,Z 352.866,A -85,B 0,C 180,E1 -17031.653,E2 -17031.653} C_VEL
LIN {X 0,Y 291.084,Z 332.914,A -85,B 0,C 180,E1 -17032.489,E2 -17032.489} C_VEL
LIN {X 0,Y 287.416,Z 314.698,A -85,B 0,C 180,E1 -17033.412,E2 -17033.412} C_VEL
LIN {X 0,Y 287.616,Z 311.389,A -85,B 0,C 180,E1 -17034.544,E2 -17034.544} C_VEL
LIN {X 0,Y 285.982,Z 302.626,A -85,B 0,C 180,E1 -17037.834,E2 -17037.834} C_VEL
LIN {X 0,Y 284.315,Z 294.88,A -85,B 0,C 180,E1 -17040.957,E2 -17040.957} C_VEL
LIN {X 0,Y 284.337,Z 294.88,A -85,B 0,C 180,E1 -17045.347,E2 -17045.347} C_VEL
LIN {X 0,Y 284.308,Z 294.888,A -85,B 0,C 180,E1 -17048.168,E2 -17048.168} C_VEL
LIN {X 0,Y 284.264,Z 294.889,A -85,B 0,C 180,E1 -17052.123,E2 -17052.123} C_VEL
LIN {X 0,Y 284.25,Z 294.892,A -85,B 0,C 180,E1 -17056.188,E2 -17056.188} C_VEL
LIN {X 0,Y 284.301,Z 294.884,A -85,B 0,C 180,E1 -17060.023,E2 -17060.023} C_VEL
LIN {X 0,Y 284.326,Z 294.874,A -85,B 0,C 180,E1 -17063.613,E2 -17063.613} C_VEL
LIN {X 0,Y 284.301,Z 294.874,A -85,B 0,C 180,E1 -17067.189,E2 -17067.189} C_VEL
LIN {X 0,Y 284.351,Z 294.875,A -85,B 0,C 180,E1 -17070.375,E2 -17070.375} C_VEL
LIN {X 0,Y 284.368,Z 294.864,A -85,B 0,C 180,E1 -17073.586,E2 -17073.586} C_VEL
LIN {X 0,Y 284.325,Z 294.874,A -85,B 0,C 180,E1 -17076.704,E2 -17076.704} C_VEL
LIN {X 0,Y 284.394,Z 294.87,A -85,B 0,C 180,E1 -17081.261,E2 -17081.261} C_VEL
LIN {X 0,Y 284.47,Z 294.847,A -85,B 0,C 180,E1 -17084.47,E2 -17084.47} C_VEL
LIN {X 0,Y 284.478,Z 294.857,A -85,B 0,C 180,E1 -17088.601,E2 -17088.601} C_VEL
LIN {X 0,Y 284.63,Z 294.83,A -85,B 0,C 180,E1 -17091.48,E2 -17091.48} C_VEL
LIN {X 0,Y 284.587,Z 294.846,A -85,B 0,C 180,E1 -17094.331,E2 -17094.331} C_VEL
LIN {X 0,Y 284.845,Z 294.809,A -85,B 0,C 180,E1 -17098.586,E2 -17098.586} C_VEL
LIN {X 0,Y 284.845,Z 294.803,A -85,B 0,C 180,E1 -17101.414,E2 -17101.414} C_VEL
LIN {X 0,Y 284.638,Z 294.832,A -85,B 0,C 180,E1 -17107.092,E2 -17107.092} C_VEL
LIN {X 0,Y 284.509,Z 294.857,A -85,B 0,C 180,E1 -17109.958,E2 -17109.958} C_VEL
LIN {X 0,Y 284.469,Z 294.863,A -85,B 0,C 180,E1 -17114.304,E2 -17114.304} C_VEL
LIN {X 0,Y 284.417,Z 294.864,A -85,B 0,C 180,E1 -17117.249,E2 -17117.249} C_VEL
LIN {X 0,Y 284.372,Z 294.871,A -85,B 0,C 180,E1 -17120.243,E2 -17120.243} C_VEL
LIN {X 0,Y 284.362,Z 294.876,A -85,B 0,C 180,E1 -17123.876,E2 -17123.876} C_VEL
LIN {X 0,Y 284.391,Z 294.871,A -85,B 0,C 180,E1 -17127.174,E2 -17127.174} C_VEL
LIN {X 0,Y 284.289,Z 294.884,A -85,B 0,C 180,E1 -17131.275,E2 -17131.275} C_VEL
LIN {X 0,Y 284.355,Z 294.874,A -85,B 0,C 180,E1 -17135.745,E2 -17135.745} C_VEL
LIN {X 0,Y 284.358,Z 295.001,A -85,B 0,C 180,E1 -17136.063,E2 -17136.063} C_VEL
LIN {X 0,Y 285.741,Z 301.185,A -85,B 0,C 180,E1 -17138.504,E2 -17138.504} C_VEL
LIN {X 0,Y 292.019,Z 316.472,A -85,B 0,C 180,E1 -17139.579,E2 -17139.579} C_VEL
LIN {X 0,Y 294.616,Z 329.937,A -85,B 0,C 180,E1 -17140.209,E2 -17140.209} C_VEL
LIN {X 0,Y 293.238,Z 378.583,A -85,B 0,C 180,E1 -17141.495,E2 -17141.495} C_VEL
LIN {X 0,Y 292.618,Z 389.648,A -85,B 0,C 180,E1 -17142.01,E2 -17142.01} C_VEL
LIN {X 0,Y 291.699,Z 401.127,A -85,B 0,C 180,E1 -17142.854,E2 -17142.854} C_VEL
LIN {X 0,Y 290.712,Z 409.82,A -85,B 0,C 180,E1 -17143.709,E2 -17143.709} C_VEL
LIN {X 0,Y 289.712,Z 417.855,A -85,B 0,C 180,E1 -17144.709,E2 -17144.709} C_VEL
LIN {X 0,Y 288.598,Z 425.113,A -85,B 0,C 180,E1 -17145.808,E2 -17145.808} C_VEL
LIN {X 0,Y 287.658,Z 430.823,A -85,B 0,C 180,E1 -17146.838,E2 -17146.838} C_VEL
LIN {X 0,Y 286.643,Z 436.621,A -85,B 0,C 180,E1 -17148.079,E2 -17148.079} C_VEL
LIN {X 0,Y 285.509,Z 442.9,A -85,B 0,C 180,E1 -17149.737,E2 -17149.737} C_VEL
LIN {X 0,Y 284.593,Z 448.027,A -85,B 0,C 180,E1 -17151.426,E2 -17151.426} C_VEL
LIN {X 0,Y 283.919,Z 451.694,A -85,B 0,C 180,E1 -17152.924,E2 -17152.924} C_VEL
LIN {X 0,Y 283.126,Z 455.57,A -85,B 0,C 180,E1 -17155.001,E2 -17155.001} C_VEL
LIN {X 0,Y 282.709,Z 457.977,A -85,B 0,C 180,E1 -17156.846,E2 -17156.846} C_VEL
LIN {X 0,Y 282.406,Z 459.366,A -85,B 0,C 180,E1 -17158.494,E2 -17158.494} C_VEL
LIN {X 0,Y 282.107,Z 460.199,A -85,B 0,C 180,E1 -17160.685,E2 -17160.685} C_VEL
LIN {X 0,Y 282.106,Z 459.59,A -85,B 0,C 180,E1 -17163.358,E2 -17163.358} C_VEL
LIN {X 0,Y 282.225,Z 458.406,A -85,B 0,C 180,E1 -17164.955,E2 -17164.955} C_VEL
LIN {X 0,Y 282.584,Z 455.908,A -85,B 0,C 180,E1 -17166.957,E2 -17166.957} C_VEL
LIN {X 0,Y 282.963,Z 452.432,A -85,B 0,C 180,E1 -17168.892,E2 -17168.892} C_VEL
LIN {X 0,Y 283.508,Z 447.784,A -85,B 0,C 180,E1 -17170.826,E2 -17170.826} C_VEL
LIN {X 0,Y 284.07,Z 443.128,A -85,B 0,C 180,E1 -17172.359,E2 -17172.359} C_VEL
LIN {X 0,Y 284.808,Z 437.308,A -85,B 0,C 180,E1 -17173.92,E2 -17173.92} C_VEL
LIN {X 0,Y 285.647,Z 430.578,A -85,B 0,C 180,E1 -17175.393,E2 -17175.393} C_VEL
LIN {X 0,Y 286.835,Z 420.844,A -85,B 0,C 180,E1 -17177.081,E2 -17177.081} C_VEL
LIN {X 0,Y 287.78,Z 412.027,A -85,B 0,C 180,E1 -17178.258,E2 -17178.258} C_VEL
LIN {X 0,Y 288.524,Z 404.002,A -85,B 0,C 180,E1 -17179.119,E2 -17179.119} C_VEL
LIN {X 0,Y 289.064,Z 395.459,A -85,B 0,C 180,E1 -17179.848,E2 -17179.848} C_VEL
LIN {X 0,Y 289.647,Z 386.04,A -85,B 0,C 180,E1 -17180.442,E2 -17180.442} C_VEL
LIN {X 0,Y 290.094,Z 376.374,A -85,B 0,C 180,E1 -17180.852,E2 -17180.852} C_VEL
LIN {X 0,Y 291.099,Z 328.415,A -85,B 0,C 180,E1 -17182.102,E2 -17182.102} C_VEL
LIN {X 0,Y 287.152,Z 306.508,A -85,B 0,C 180,E1 -17182.941,E2 -17182.941} C_VEL
LIN {X 0,Y 285.656,Z 301.023,A -85,B 0,C 180,E1 -17183.2,E2 -17183.2} C_VEL
LIN {X 0,Y 284.527,Z 294.86,A -85,B 0,C 180,E1 -17185.751,E2 -17185.751} C_VEL
LIN {X 0,Y 284.856,Z 294.814,A -85,B 0,C 180,E1 -17188.586,E2 -17188.586} C_VEL
LIN {X 0,Y 284.856,Z 294.814,A -85,B 0,C 180,E1 -17191.414,E2 -17191.414} C_VEL
LIN {X 0,Y 284.656,Z 294.836,A -85,B 0,C 180,E1 -17197.091,E2 -17197.091} C_VEL
LIN {X 0,Y 284.519,Z 294.857,A -85,B 0,C 180,E1 -17199.957,E2 -17199.957} C_VEL
LIN {X 0,Y 284.464,Z 294.863,A -85,B 0,C 180,E1 -17204.303,E2 -17204.303} C_VEL
LIN {X 0,Y 284.375,Z 294.872,A -85,B 0,C 180,E1 -17208.74,E2 -17208.74} C_VEL
LIN {X 0,Y 284.312,Z 294.871,A -85,B 0,C 180,E1 -17211.764,E2 -17211.764} C_VEL
LIN {X 0,Y 284.336,Z 294.88,A -85,B 0,C 180,E1 -17214.846,E2 -17214.846} C_VEL
LIN {X 0,Y 284.33,Z 294.878,A -85,B 0,C 180,E1 -17218.01,E2 -17218.01} C_VEL
LIN {X 0,Y 284.294,Z 294.883,A -85,B 0,C 180,E1 -17221.273,E2 -17221.273} C_VEL
LIN {X 0,Y 284.339,Z 294.88,A -85,B 0,C 180,E1 -17225.347,E2 -17225.347} C_VEL
LIN {X 0,Y 284.306,Z 294.88,A -85,B 0,C 180,E1 -17228.169,E2 -17228.169} C_VEL
LIN {X 0,Y 284.28,Z 294.879,A -85,B 0,C 180,E1 -17232.126,E2 -17232.126} C_VEL
LIN {X 0,Y 284.314,Z 294.879,A -85,B 0,C 180,E1 -17236.2,E2 -17236.2} C_VEL
LIN {X 0,Y 284.347,Z 294.877,A -85,B 0,C 180,E1 -17240.012,E2 -17240.012} C_VEL
LIN {X 0,Y 284.347,Z 294.876,A -85,B 0,C 180,E1 -17243.616,E2 -17243.616} C_VEL
LIN {X 0,Y 284.302,Z 294.878,A -85,B 0,C 180,E1 -17247.189,E2 -17247.189} C_VEL
LIN {X 0,Y 284.352,Z 294.877,A -85,B 0,C 180,E1 -17250.375,E2 -17250.375} C_VEL
LIN {X 0,Y 284.372,Z 294.872,A -85,B 0,C 180,E1 -17253.586,E2 -17253.586} C_VEL
LIN {X 0,Y 284.359,Z 294.871,A -85,B 0,C 180,E1 -17256.706,E2 -17256.706} C_VEL
LIN {X 0,Y 284.395,Z 294.865,A -85,B 0,C 180,E1 -17261.261,E2 -17261.261} C_VEL
LIN {X 0,Y 284.471,Z 294.863,A -85,B 0,C 180,E1 -17264.469,E2 -17264.469} C_VEL
LIN {X 0,Y 284.479,Z 294.863,A -85,B 0,C 180,E1 -17268.601,E2 -17268.601} C_VEL
LIN {X 0,Y 284.487,Z 294.856,A -85,B 0,C 180,E1 -17269.706,E2 -17269.706} C_VEL
LIN {X 0,Y 283.848,Z 294.939,A -85,B 0,C 180,E1 -17270.889,E2 -17270.889} C_VEL
LIN {X 0,Y 280.938,Z 295.299,A -85,B 0,C 180,E1 -17272.814,E2 -17272.814} C_VEL
LIN {X 0,Y 278.498,Z 295.599,A -85,B 0,C 180,E1 -17274.379,E2 -17274.379} C_VEL
LIN {X 0,Y 277.529,Z 295.719,A -85,B 0,C 180,E1 -17275.593,E2 -17275.593} C_VEL
LIN {X 0,Y 277.494,Z 295.722,A -85,B 0,C 180,E1 -17276.004,E2 -17276.004} C_VEL
LIN {X 0,Y 277.812,Z 295.687,A -85,B 0,C 180,E1 -17278.55,E2 -17278.55} C_VEL
LIN {X 0,Y 277.813,Z 295.691,A -85,B 0,C 180,E1 -17281.449,E2 -17281.449} C_VEL
LIN {X 0,Y 277.631,Z 295.713,A -85,B 0,C 180,E1 -17287.271,E2 -17287.271} C_VEL
LIN {X 0,Y 277.454,Z 295.729,A -85,B 0,C 180,E1 -17290.213,E2 -17290.213} C_VEL
LIN {X 0,Y 277.42,Z 295.737,A -85,B 0,C 180,E1 -17294.675,E2 -17294.675} C_VEL
LIN {X 0,Y 277.334,Z 295.748,A -85,B 0,C 180,E1 -17299.234,E2 -17299.234} C_VEL
LIN {X 0,Y 277.285,Z 295.758,A -85,B 0,C 180,E1 -17304.158,E2 -17304.158} C_VEL
LIN {X 0,Y 277.316,Z 295.752,A -85,B 0,C 180,E1 -17307.505,E2 -17307.505} C_VEL
LIN {X 0,Y 277.266,Z 295.758,A -85,B 0,C 180,E1 -17310.482,E2 -17310.482} C_VEL
LIN {X 0,Y 277.241,Z 295.762,A -85,B 0,C 180,E1 -17313.896,E2 -17313.896} C_VEL
LIN {X 0,Y 277.261,Z 295.756,A -85,B 0,C 180,E1 -17317.47,E2 -17317.47} C_VEL
LIN {X 0,Y 277.204,Z 295.759,A -85,B 0,C 180,E1 -17321.237,E2 -17321.237} C_VEL
LIN {X 0,Y 277.212,Z 295.765,A -85,B 0,C 180,E1 -17325.224,E2 -17325.224} C_VEL
LIN {X 0,Y 277.218,Z 295.764,A -85,B 0,C 180,E1 -17329.513,E2 -17329.513} C_VEL
LIN {X 0,Y 277.261,Z 295.76,A -85,B 0,C 180,E1 -17332.531,E2 -17332.531} C_VEL
LIN {X 0,Y 277.243,Z 295.76,A -85,B 0,C 180,E1 -17336.105,E2 -17336.105} C_VEL
LIN {X 0,Y 277.313,Z 295.816,A -85,B 0,C 180,E1 -17340.957,E2 -17340.957} C_VEL
LIN {X 0,Y 279.26,Z 306.187,A -85,B 0,C 180,E1 -17344.957,E2 -17344.957} C_VEL
LIN {X 0,Y 279.718,Z 309.797,A -85,B 0,C 180,E1 -17346.297,E2 -17346.297} C_VEL
LIN {X 0,Y 278.97,Z 315.76,A -85,B 0,C 180,E1 -17348.391,E2 -17348.391} C_VEL
LIN {X 0,Y 283.862,Z 352.631,A -85,B 0,C 180,E1 -17349.735,E2 -17349.735} C_VEL
LIN {X 0,Y 283.047,Z 393.352,A -85,B 0,C 180,E1 -17350.847,E2 -17350.847} C_VEL
LIN {X 0,Y 282.362,Z 404.273,A -85,B 0,C 180,E1 -17351.357,E2 -17351.357} C_VEL
LIN {X 0,Y 281.51,Z 415.629,A -85,B 0,C 180,E1 -17352.193,E2 -17352.193} C_VEL
LIN {X 0,Y 280.621,Z 424.452,A -85,B 0,C 180,E1 -17353.074,E2 -17353.074} C_VEL
LIN {X 0,Y 279.717,Z 432.875,A -85,B 0,C 180,E1 -17354.143,E2 -17354.143} C_VEL
LIN {X 0,Y 278.745,Z 440.834,A -85,B 0,C 180,E1 -17355.397,E2 -17355.397} C_VEL
LIN {X 0,Y 277.802,Z 448.272,A -85,B 0,C 180,E1 -17356.839,E2 -17356.839} C_VEL
LIN {X 0,Y 276.862,Z 455.811,A -85,B 0,C 180,E1 -17358.655,E2 -17358.655} C_VEL
LIN {X 0,Y 276.178,Z 461.714,A -85,B 0,C 180,E1 -17360.479,E2 -17360.479} C_VEL
LIN {X 0,Y 275.749,Z 465.549,A -85,B 0,C 180,E1 -17361.942,E2 -17361.942} C_VEL
LIN {X 0,Y 275.414,Z 469.943,A -85,B 0,C 180,E1 -17364.142,E2 -17364.142} C_VEL
LIN {X 0,Y 275.281,Z 472.189,A -85,B 0,C 180,E1 -17365.607,E2 -17365.607} C_VEL
LIN {X 0,Y 275.285,Z 473.819,A -85,B 0,C 180,E1 -17367.073,E2 -17367.073} C_VEL
LIN {X 0,Y 275.259,Z 474.869,A -85,B 0,C 180,E1 -17368.537,E2 -17368.537} C_VEL
LIN {X 0,Y 275.275,Z 475.439,A -85,B 0,C 180,E1 -17370,E2 -17370} C_VEL
LIN {X 0,Y 275.256,Z 475.538,A -85,B 0,C 180,E1 -17371.463,E2 -17371.463} C_VEL
LIN {X 0,Y 275.267,Z 475.152,A -85,B 0,C 180,E1 -17372.927,E2 -17372.927} C_VEL
LIN {X 0,Y 275.334,Z 473.142,A -85,B 0,C 180,E1 -17375.447,E2 -17375.447} C_VEL
LIN {X 0,Y 275.644,Z 470.676,A -85,B 0,C 180,E1 -17377.324,E2 -17377.324} C_VEL
LIN {X 0,Y 276.312,Z 466.593,A -85,B 0,C 180,E1 -17379.516,E2 -17379.516} C_VEL
LIN {X 0,Y 277.247,Z 461.101,A -85,B 0,C 180,E1 -17381.7,E2 -17381.7} C_VEL
LIN {X 0,Y 278.431,Z 455.106,A -85,B 0,C 180,E1 -17383.502,E2 -17383.502} C_VEL
LIN {X 0,Y 279.464,Z 449.252,A -85,B 0,C 180,E1 -17384.937,E2 -17384.937} C_VEL
LIN {X 0,Y 280.713,Z 442.138,A -85,B 0,C 180,E1 -17386.359,E2 -17386.359} C_VEL
LIN {X 0,Y 281.981,Z 434.578,A -85,B 0,C 180,E1 -17387.589,E2 -17387.589} C_VEL
LIN {X 0,Y 283.233,Z 426.695,A -85,B 0,C 180,E1 -17388.63,E2 -17388.63} C_VEL
LIN {X 0,Y 284.183,Z 418.634,A -85,B 0,C 180,E1 -17389.503,E2 -17389.503} C_VEL
LIN {X 0,Y 285.222,Z 409.25,A -85,B 0,C 180,E1 -17390.281,E2 -17390.281} C_VEL
LIN {X 0,Y 286.136,Z 399.675,A -85,B 0,C 180,E1 -17390.854,E2 -17390.854} C_VEL
LIN {X 0,Y 286.784,Z 388.191,A -85,B 0,C 180,E1 -17391.306,E2 -17391.306} C_VEL
LIN {X 0,Y 287.569,Z 353.763,A -85,B 0,C 180,E1 -17392.225,E2 -17392.225} C_VEL
LIN {X 0,Y 285.054,Z 335.855,A -85,B 0,C 180,E1 -17392.995,E2 -17392.995} C_VEL
LIN {X 0,Y 280.692,Z 314.593,A -85,B 0,C 180,E1 -17394.08,E2 -17394.08} C_VEL
LIN {X 0,Y 280.379,Z 310.655,A -85,B 0,C 180,E1 -17395.528,E2 -17395.528} C_VEL
LIN {X 0,Y 278.359,Z 300.579,A -85,B 0,C 180,E1 -17399.493,E2 -17399.493} C_VEL
LIN {X 0,Y 277.256,Z 295.758,A -85,B 0,C 180,E1 -17401.519,E2 -17401.519} C_VEL
LIN {X 0,Y 277.277,Z 295.761,A -85,B 0,C 180,E1 -17405.798,E2 -17405.798} C_VEL
LIN {X 0,Y 277.23,Z 295.768,A -85,B 0,C 180,E1 -17409.327,E2 -17409.327} C_VEL
LIN {X 0,Y 277.205,Z 295.774,A -85,B 0,C 180,E1 -17413.197,E2 -17413.197} C_VEL
LIN {X 0,Y 277.209,Z 295.77,A -85,B 0,C 180,E1 -17417.324,E2 -17417.324} C_VEL
LIN {X 0,Y 277.259,Z 295.756,A -85,B 0,C 180,E1 -17421.792,E2 -17421.792} C_VEL
LIN {X 0,Y 277.278,Z 295.758,A -85,B 0,C 180,E1 -17424.341,E2 -17424.341} C_VEL
LIN {X 0,Y 277.238,Z 295.753,A -85,B 0,C 180,E1 -17427.836,E2 -17427.836} C_VEL
LIN {X 0,Y 277.282,Z 295.754,A -85,B 0,C 180,E1 -17431.212,E2 -17431.212} C_VEL
LIN {X 0,Y 277.301,Z 295.754,A -85,B 0,C 180,E1 -17434.478,E2 -17434.478} C_VEL
LIN {X 0,Y 277.26,Z 295.748,A -85,B 0,C 180,E1 -17437.653,E2 -17437.653} C_VEL
LIN {X 0,Y 277.336,Z 295.751,A -85,B 0,C 180,E1 -17440.766,E2 -17440.766} C_VEL
LIN {X 0,Y 277.42,Z 295.729,A -85,B 0,C 180,E1 -17445.325,E2 -17445.325} C_VEL
LIN {X 0,Y 277.452,Z 295.725,A -85,B 0,C 180,E1 -17449.787,E2 -17449.787} C_VEL
LIN {X 0,Y 277.631,Z 295.709,A -85,B 0,C 180,E1 -17452.729,E2 -17452.729} C_VEL
LIN {X 0,Y 277.811,Z 295.685,A -85,B 0,C 180,E1 -17458.551,E2 -17458.551} C_VEL
LIN {X 0,Y 277.811,Z 295.679,A -85,B 0,C 180,E1 -17461.45,E2 -17461.45} C_VEL
LIN {X 0,Y 277.596,Z 295.708,A -85,B 0,C 180,E1 -17467.273,E2 -17467.273} C_VEL
LIN {X 0,Y 277.452,Z 295.736,A -85,B 0,C 180,E1 -17470.214,E2 -17470.214} C_VEL
LIN {X 0,Y 277.42,Z 295.741,A -85,B 0,C 180,E1 -17474.675,E2 -17474.675} C_VEL
LIN {X 0,Y 277.337,Z 295.756,A -85,B 0,C 180,E1 -17479.235,E2 -17479.235} C_VEL
LIN {X 0,Y 277.312,Z 295.754,A -85,B 0,C 180,E1 -17484.171,E2 -17484.171} C_VEL
LIN {X 0,Y 277.32,Z 295.753,A -85,B 0,C 180,E1 -17487.506,E2 -17487.506} C_VEL
LIN {X 0,Y 277.266,Z 295.759,A -85,B 0,C 180,E1 -17490.482,E2 -17490.482} C_VEL
LIN {X 0,Y 277.316,Z 295.748,A -85,B 0,C 180,E1 -17495.32,E2 -17495.32} C_VEL
LIN {X 0,Y 278.36,Z 300.255,A -85,B 0,C 180,E1 -17497.297,E2 -17497.297} C_VEL
LIN {X 0,Y 278.626,Z 301.45,A -85,B 0,C 180,E1 -17497.742,E2 -17497.742} C_VEL
LIN {X 0,Y 285.917,Z 318.86,A -85,B 0,C 180,E1 -17499.041,E2 -17499.041} C_VEL
LIN {X 0,Y 288.257,Z 331.092,A -85,B 0,C 180,E1 -17499.632,E2 -17499.632} C_VEL
LIN {X 0,Y 286.781,Z 378.652,A -85,B 0,C 180,E1 -17500.914,E2 -17500.914} C_VEL
LIN {X 0,Y 286.146,Z 389.372,A -85,B 0,C 180,E1 -17501.418,E2 -17501.418} C_VEL
LIN {X 0,Y 285.159,Z 401.483,A -85,B 0,C 180,E1 -17502.324,E2 -17502.324} C_VEL
LIN {X 0,Y 284.166,Z 409.744,A -85,B 0,C 180,E1 -17503.15,E2 -17503.15} C_VEL
LIN {X 0,Y 283.116,Z 417.628,A -85,B 0,C 180,E1 -17504.141,E2 -17504.141} C_VEL
LIN {X 0,Y 282.002,Z 424.85,A -85,B 0,C 180,E1 -17505.25,E2 -17505.25} C_VEL
LIN {X 0,Y 280.757,Z 431.813,A -85,B 0,C 180,E1 -17506.547,E2 -17506.547} C_VEL
LIN {X 0,Y 279.74,Z 437.314,A -85,B 0,C 180,E1 -17507.776,E2 -17507.776} C_VEL
LIN {X 0,Y 278.535,Z 443.738,A -85,B 0,C 180,E1 -17509.546,E2 -17509.546} C_VEL
LIN {X 0,Y 277.784,Z 447.423,A -85,B 0,C 180,E1 -17510.766,E2 -17510.766} C_VEL
LIN {X 0,Y 276.992,Z 451.643,A -85,B 0,C 180,E1 -17512.488,E2 -17512.488} C_VEL
LIN {X 0,Y 276.158,Z 455.44,A -85,B 0,C 180,E1 -17514.526,E2 -17514.526} C_VEL
LIN {X 0,Y 275.865,Z 457.391,A -85,B 0,C 180,E1 -17515.913,E2 -17515.913} C_VEL
LIN {X 0,Y 275.477,Z 459.106,A -85,B 0,C 180,E1 -17517.606,E2 -17517.606} C_VEL
LIN {X 0,Y 275.189,Z 460.129,A -85,B 0,C 180,E1 -17519.286,E2 -17519.286} C_VEL
LIN {X 0,Y 275.016,Z 460.465,A -85,B 0,C 180,E1 -17520.953,E2 -17520.953} C_VEL
LIN {X 0,Y 275.013,Z 459.703,A -85,B 0,C 180,E1 -17523.436,E2 -17523.436} C_VEL
LIN {X 0,Y 275.296,Z 457.54,A -85,B 0,C 180,E1 -17525.893,E2 -17525.893} C_VEL
LIN {X 0,Y 275.612,Z 455.284,A -85,B 0,C 180,E1 -17527.513,E2 -17527.513} C_VEL
LIN {X 0,Y 275.935,Z 452.362,A -85,B 0,C 180,E1 -17529.111,E2 -17529.111} C_VEL
LIN {X 0,Y 276.386,Z 448.692,A -85,B 0,C 180,E1 -17530.697,E2 -17530.697} C_VEL
LIN {X 0,Y 276.928,Z 444.196,A -85,B 0,C 180,E1 -17532.27,E2 -17532.27} C_VEL
LIN {X 0,Y 277.75,Z 437.832,A -85,B 0,C 180,E1 -17534.055,E2 -17534.055} C_VEL
LIN {X 0,Y 278.737,Z 430.193,A -85,B 0,C 180,E1 -17535.769,E2 -17535.769} C_VEL
LIN {X 0,Y 279.984,Z 420.215,A -85,B 0,C 180,E1 -17537.495,E2 -17537.495} C_VEL
LIN {X 0,Y 280.932,Z 411.727,A -85,B 0,C 180,E1 -17538.638,E2 -17538.638} C_VEL
LIN {X 0,Y 281.737,Z 402.938,A -85,B 0,C 180,E1 -17539.581,E2 -17539.581} C_VEL
LIN {X 0,Y 282.34,Z 393.996,A -85,B 0,C 180,E1 -17540.328,E2 -17540.328} C_VEL
LIN {X 0,Y 282.915,Z 384.03,A -85,B 0,C 180,E1 -17540.933,E2 -17540.933} C_VEL
LIN {X 0,Y 283.379,Z 371.521,A -85,B 0,C 180,E1 -17541.398,E2 -17541.398} C_VEL
LIN {X 0,Y 284.307,Z 329.18,A -85,B 0,C 180,E1 -17542.501,E2 -17542.501} C_VEL
LIN {X 0,Y 280.45,Z 307.956,A -85,B 0,C 180,E1 -17543.345,E2 -17543.345} C_VEL
LIN {X 0,Y 278.601,Z 301.247,A -85,B 0,C 180,E1 -17543.664,E2 -17543.664} C_VEL
LIN {X 0,Y 277.509,Z 295.734,A -85,B 0,C 180,E1 -17546.007,E2 -17546.007} C_VEL
LIN {X 0,Y 277.822,Z 295.691,A -85,B 0,C 180,E1 -17548.551,E2 -17548.551} C_VEL
LIN {X 0,Y 277.822,Z 295.69,A -85,B 0,C 180,E1 -17551.45,E2 -17551.45} C_VEL
LIN {X 0,Y 277.614,Z 295.713,A -85,B 0,C 180,E1 -17557.272,E2 -17557.272} C_VEL
LIN {X 0,Y 277.462,Z 295.737,A -85,B 0,C 180,E1 -17560.213,E2 -17560.213} C_VEL
LIN {X 0,Y 277.411,Z 295.742,A -85,B 0,C 180,E1 -17564.675,E2 -17564.675} C_VEL
LIN {X 0,Y 277.324,Z 295.747,A -85,B 0,C 180,E1 -17569.235,E2 -17569.235} C_VEL
LIN {X 0,Y 277.291,Z 295.751,A -85,B 0,C 180,E1 -17574.157,E2 -17574.157} C_VEL
LIN {X 0,Y 277.324,Z 295.752,A -85,B 0,C 180,E1 -17577.504,E2 -17577.504} C_VEL
LIN {X 0,Y 277.271,Z 295.759,A -85,B 0,C 180,E1 -17580.48,E2 -17580.48} C_VEL
LIN {X 0,Y 277.245,Z 295.759,A -85,B 0,C 180,E1 -17583.895,E2 -17583.895} C_VEL
LIN {X 0,Y 277.263,Z 295.761,A -85,B 0,C 180,E1 -17587.469,E2 -17587.469} C_VEL
LIN {X 0,Y 277.212,Z 295.766,A -85,B 0,C 180,E1 -17591.234,E2 -17591.234} C_VEL
LIN {X 0,Y 277.243,Z 295.76,A -85,B 0,C 180,E1 -17595.216,E2 -17595.216} C_VEL
LIN {X 0,Y 277.291,Z 295.758,A -85,B 0,C 180,E1 -17599.494,E2 -17599.494} C_VEL
LIN {X 0,Y 277.281,Z 295.752,A -85,B 0,C 180,E1 -17602.533,E2 -17602.533} C_VEL
LIN {X 0,Y 277.249,Z 295.759,A -85,B 0,C 180,E1 -17606.104,E2 -17606.104} C_VEL
LIN {X 0,Y 277.256,Z 295.758,A -85,B 0,C 180,E1 -17609.538,E2 -17609.538} C_VEL
LIN {X 0,Y 277.353,Z 295.746,A -85,B 0,C 180,E1 -17612.863,E2 -17612.863} C_VEL
LIN {X 0,Y 277.322,Z 295.752,A -85,B 0,C 180,E1 -17616.079,E2 -17616.079} C_VEL
LIN {X 0,Y 277.337,Z 295.746,A -85,B 0,C 180,E1 -17620.765,E2 -17620.765} C_VEL
LIN {X 0,Y 277.42,Z 295.738,A -85,B 0,C 180,E1 -17625.325,E2 -17625.325} C_VEL
LIN {X 0,Y 277.453,Z 295.733,A -85,B 0,C 180,E1 -17629.787,E2 -17629.787} C_VEL
LIN {X 0,Y 277.632,Z 295.712,A -85,B 0,C 180,E1 -17632.728,E2 -17632.728} C_VEL
LIN {X 0,Y 277.494,Z 295.722,A -85,B 0,C 180,E1 -17636.004,E2 -17636.004} C_VEL
LIN {X 0,Y 276.973,Z 295.794,A -85,B 0,C 180,E1 -17637.219,E2 -17637.219} C_VEL
LIN {X 0,Y 274.263,Z 296.134,A -85,B 0,C 180,E1 -17639.201,E2 -17639.201} C_VEL
LIN {X 0,Y 271.019,Z 296.536,A -85,B 0,C 180,E1 -17641.638,E2 -17641.638} C_VEL
LIN {X 0,Y 270.652,Z 296.581,A -85,B 0,C 180,E1 -17642.48,E2 -17642.48} C_VEL
LIN {X 0,Y 270.59,Z 296.587,A -85,B 0,C 180,E1 -17647.462,E2 -17647.462} C_VEL
LIN {X 0,Y 270.406,Z 296.606,A -85,B 0,C 180,E1 -17650.482,E2 -17650.482} C_VEL
LIN {X 0,Y 270.389,Z 296.614,A -85,B 0,C 180,E1 -17655.065,E2 -17655.065} C_VEL
LIN {X 0,Y 270.292,Z 296.627,A -85,B 0,C 180,E1 -17659.756,E2 -17659.756} C_VEL
LIN {X 0,Y 270.231,Z 296.634,A -85,B 0,C 180,E1 -17664.59,E2 -17664.59} C_VEL
LIN {X 0,Y 270.263,Z 296.633,A -85,B 0,C 180,E1 -17667.909,E2 -17667.909} C_VEL
LIN {X 0,Y 270.178,Z 296.638,A -85,B 0,C 180,E1 -17671.349,E2 -17671.349} C_VEL
LIN {X 0,Y 270.196,Z 296.64,A -85,B 0,C 180,E1 -17674.906,E2 -17674.906} C_VEL
LIN {X 0,Y 270.192,Z 296.636,A -85,B 0,C 180,E1 -17678.711,E2 -17678.711} C_VEL
LIN {X 0,Y 270.167,Z 296.64,A -85,B 0,C 180,E1 -17683.251,E2 -17683.251} C_VEL
LIN {X 0,Y 270.17,Z 296.642,A -85,B 0,C 180,E1 -17687.443,E2 -17687.443} C_VEL
LIN {X 0,Y 270.204,Z 296.639,A -85,B 0,C 180,E1 -17691.375,E2 -17691.375} C_VEL
LIN {X 0,Y 270.198,Z 296.642,A -85,B 0,C 180,E1 -17695.095,E2 -17695.095} C_VEL
LIN {X 0,Y 270.181,Z 296.645,A -85,B 0,C 180,E1 -17699.137,E2 -17699.137} C_VEL
LIN {X 0,Y 270.264,Z 296.728,A -85,B 0,C 180,E1 -17700.673,E2 -17700.673} C_VEL
LIN {X 0,Y 272.159,Z 306.799,A -85,B 0,C 180,E1 -17704.663,E2 -17704.663} C_VEL
LIN {X 0,Y 272.675,Z 310.426,A -85,B 0,C 180,E1 -17706.05,E2 -17706.05} C_VEL
LIN {X 0,Y 272.047,Z 315.514,A -85,B 0,C 180,E1 -17707.888,E2 -17707.888} C_VEL
LIN {X 0,Y 276.711,Z 350.451,A -85,B 0,C 180,E1 -17709.228,E2 -17709.228} C_VEL
LIN {X 0,Y 277.107,Z 356.252,A -85,B 0,C 180,E1 -17709.416,E2 -17709.416} C_VEL
LIN {X 0,Y 276.246,Z 392.93,A -85,B 0,C 180,E1 -17710.44,E2 -17710.44} C_VEL
LIN {X 0,Y 275.629,Z 403.351,A -85,B 0,C 180,E1 -17710.932,E2 -17710.932} C_VEL
LIN {X 0,Y 274.997,Z 411.113,A -85,B 0,C 180,E1 -17711.467,E2 -17711.467} C_VEL
LIN {X 0,Y 273.981,Z 421.975,A -85,B 0,C 180,E1 -17712.459,E2 -17712.459} C_VEL
LIN {X 0,Y 272.873,Z 432.092,A -85,B 0,C 180,E1 -17713.735,E2 -17713.735} C_VEL
LIN {X 0,Y 271.876,Z 440.152,A -85,B 0,C 180,E1 -17715.019,E2 -17715.019} C_VEL
LIN {X 0,Y 271.146,Z 445.953,A -85,B 0,C 180,E1 -17716.128,E2 -17716.128} C_VEL
LIN {X 0,Y 270.286,Z 452.418,A -85,B 0,C 180,E1 -17717.613,E2 -17717.613} C_VEL
LIN {X 0,Y 269.527,Z 457.782,A -85,B 0,C 180,E1 -17719.103,E2 -17719.103} C_VEL
LIN {X 0,Y 268.915,Z 463.222,A -85,B 0,C 180,E1 -17720.979,E2 -17720.979} C_VEL
LIN {X 0,Y 268.544,Z 466.739,A -85,B 0,C 180,E1 -17722.481,E2 -17722.481} C_VEL
LIN {X 0,Y 268.232,Z 470.634,A -85,B 0,C 180,E1 -17724.65,E2 -17724.65} C_VEL
LIN {X 0,Y 268.196,Z 471.887,A -85,B 0,C 180,E1 -17725.491,E2 -17725.491} C_VEL
LIN {X 0,Y 268.196,Z 473.528,A -85,B 0,C 180,E1 -17726.996,E2 -17726.996} C_VEL
LIN {X 0,Y 268.186,Z 474.617,A -85,B 0,C 180,E1 -17728.498,E2 -17728.498} C_VEL
LIN {X 0,Y 268.199,Z 475.224,A -85,B 0,C 180,E1 -17730,E2 -17730} C_VEL
LIN {X 0,Y 268.183,Z 475.359,A -85,B 0,C 180,E1 -17731.502,E2 -17731.502} C_VEL
LIN {X 0,Y 268.18,Z 474.99,A -85,B 0,C 180,E1 -17733.004,E2 -17733.004} C_VEL
LIN {X 0,Y 268.233,Z 473.297,A -85,B 0,C 180,E1 -17735.353,E2 -17735.353} C_VEL
LIN {X 0,Y 268.801,Z 469.433,A -85,B 0,C 180,E1 -17738.268,E2 -17738.268} C_VEL
LIN {X 0,Y 269.583,Z 464.98,A -85,B 0,C 180,E1 -17740.514,E2 -17740.514} C_VEL
LIN {X 0,Y 270.517,Z 460.039,A -85,B 0,C 180,E1 -17742.376,E2 -17742.376} C_VEL
LIN {X 0,Y 271.768,Z 453.814,A -85,B 0,C 180,E1 -17744.221,E2 -17744.221} C_VEL
LIN {X 0,Y 272.922,Z 447.755,A -85,B 0,C 180,E1 -17745.687,E2 -17745.687} C_VEL
LIN {X 0,Y 274.318,Z 440.398,A -85,B 0,C 180,E1 -17747.135,E2 -17747.135} C_VEL
LIN {X 0,Y 275.682,Z 432.542,A -85,B 0,C 180,E1 -17748.389,E2 -17748.389} C_VEL
LIN {X 0,Y 276.944,Z 424.272,A -85,B 0,C 180,E1 -17749.455,E2 -17749.455} C_VEL
LIN {X 0,Y 278.259,Z 413.792,A -85,B 0,C 180,E1 -17750.514,E2 -17750.514} C_VEL
LIN {X 0,Y 279.477,Z 402.082,A -85,B 0,C 180,E1 -17751.318,E2 -17751.318} C_VEL
LIN {X 0,Y 280.113,Z 393.139,A -85,B 0,C 180,E1 -17751.738,E2 -17751.738} C_VEL
LIN {X 0,Y 281.223,Z 354.884,A -85,B 0,C 180,E1 -17752.816,E2 -17752.816} C_VEL
LIN {X 0,Y 278.659,Z 336.906,A -85,B 0,C 180,E1 -17753.621,E2 -17753.621} C_VEL
LIN {X 0,Y 274.89,Z 318.2,A -85,B 0,C 180,E1 -17754.61,E2 -17754.61} C_VEL
LIN {X 0,Y 273.796,Z 314.309,A -85,B 0,C 180,E1 -17754.874,E2 -17754.874} C_VEL
LIN {X 0,Y 272.085,Z 305.014,A -85,B 0,C 180,E1 -17758.571,E2 -17758.571} C_VEL
LIN {X 0,Y 270.2,Z 296.639,A -85,B 0,C 180,E1 -17762.167,E2 -17762.167} C_VEL
LIN {X 0,Y 270.214,Z 296.641,A -85,B 0,C 180,E1 -17766.74,E2 -17766.74} C_VEL
LIN {X 0,Y 270.165,Z 296.652,A -85,B 0,C 180,E1 -17771.027,E2 -17771.027} C_VEL
LIN {X 0,Y 270.147,Z 296.646,A -85,B 0,C 180,E1 -17775.379,E2 -17775.379} C_VEL
LIN {X 0,Y 270.168,Z 296.64,A -85,B 0,C 180,E1 -17779.433,E2 -17779.433} C_VEL
LIN {X 0,Y 270.235,Z 296.63,A -85,B 0,C 180,E1 -17783.725,E2 -17783.725} C_VEL
LIN {X 0,Y 270.196,Z 296.632,A -85,B 0,C 180,E1 -17786.892,E2 -17786.892} C_VEL
LIN {X 0,Y 270.222,Z 296.635,A -85,B 0,C 180,E1 -17790.386,E2 -17790.386} C_VEL
LIN {X 0,Y 270.253,Z 296.623,A -85,B 0,C 180,E1 -17793.763,E2 -17793.763} C_VEL
LIN {X 0,Y 270.202,Z 296.632,A -85,B 0,C 180,E1 -17797.036,E2 -17797.036} C_VEL
LIN {X 0,Y 270.293,Z 296.624,A -85,B 0,C 180,E1 -17800.244,E2 -17800.244} C_VEL
LIN {X 0,Y 270.388,Z 296.602,A -85,B 0,C 180,E1 -17804.935,E2 -17804.935} C_VEL
LIN {X 0,Y 270.404,Z 296.605,A -85,B 0,C 180,E1 -17809.518,E2 -17809.518} C_VEL
LIN {X 0,Y 270.59,Z 296.584,A -85,B 0,C 180,E1 -17812.538,E2 -17812.538} C_VEL
LIN {X 0,Y 270.777,Z 296.561,A -85,B 0,C 180,E1 -17818.513,E2 -17818.513} C_VEL
LIN {X 0,Y 270.777,Z 296.555,A -85,B 0,C 180,E1 -17821.487,E2 -17821.487} C_VEL
LIN {X 0,Y 270.557,Z 296.584,A -85,B 0,C 180,E1 -17827.463,E2 -17827.463} C_VEL
LIN {X 0,Y 270.404,Z 296.614,A -85,B 0,C 180,E1 -17830.483,E2 -17830.483} C_VEL
LIN {X 0,Y 270.389,Z 296.619,A -85,B 0,C 180,E1 -17835.066,E2 -17835.066} C_VEL
LIN {X 0,Y 270.294,Z 296.627,A -85,B 0,C 180,E1 -17839.756,E2 -17839.756} C_VEL
LIN {X 0,Y 270.268,Z 296.634,A -85,B 0,C 180,E1 -17844.586,E2 -17844.586} C_VEL
LIN {X 0,Y 270.265,Z 296.635,A -85,B 0,C 180,E1 -17847.91,E2 -17847.91} C_VEL
LIN {X 0,Y 270.179,Z 296.642,A -85,B 0,C 180,E1 -17851.349,E2 -17851.349} C_VEL
LIN {X 0,Y 270.258,Z 296.716,A -85,B 0,C 180,E1 -17854.811,E2 -17854.811} C_VEL
LIN {X 0,Y 271.386,Z 301.565,A -85,B 0,C 180,E1 -17856.904,E2 -17856.904} C_VEL
LIN {X 0,Y 279.431,Z 320.25,A -85,B 0,C 180,E1 -17858.407,E2 -17858.407} C_VEL
LIN {X 0,Y 281.478,Z 329.853,A -85,B 0,C 180,E1 -17858.911,E2 -17858.911} C_VEL
LIN {X 0,Y 281.86,Z 333.49,A -85,B 0,C 180,E1 -17859.059,E2 -17859.059} C_VEL
LIN {X 0,Y 280.374,Z 378.538,A -85,B 0,C 180,E1 -17860.297,E2 -17860.297} C_VEL
LIN {X 0,Y 279.736,Z 388.881,A -85,B 0,C 180,E1 -17860.785,E2 -17860.785} C_VEL
LIN {X 0,Y 278.749,Z 400.954,A -85,B 0,C 180,E1 -17861.677,E2 -17861.677} C_VEL
LIN {X 0,Y 277.713,Z 409.361,A -85,B 0,C 180,E1 -17862.521,E2 -17862.521} C_VEL
LIN {X 0,Y 276.445,Z 418.267,A -85,B 0,C 180,E1 -17863.665,E2 -17863.665} C_VEL
LIN {X 0,Y 275.246,Z 425.59,A -85,B 0,C 180,E1 -17864.83,E2 -17864.83} C_VEL
LIN {X 0,Y 273.944,Z 432.476,A -85,B 0,C 180,E1 -17866.159,E2 -17866.159} C_VEL
LIN {X 0,Y 272.855,Z 438.056,A -85,B 0,C 180,E1 -17867.46,E2 -17867.46} C_VEL
LIN {X 0,Y 271.713,Z 443.75,A -85,B 0,C 180,E1 -17869.072,E2 -17869.072} C_VEL
LIN {X 0,Y 270.845,Z 447.881,A -85,B 0,C 180,E1 -17870.486,E2 -17870.486} C_VEL
LIN {X 0,Y 269.991,Z 452.116,A -85,B 0,C 180,E1 -17872.288,E2 -17872.288} C_VEL
LIN {X 0,Y 269.216,Z 455.308,A -85,B 0,C 180,E1 -17874.025,E2 -17874.025} C_VEL
LIN {X 0,Y 268.804,Z 457.731,A -85,B 0,C 180,E1 -17875.798,E2 -17875.798} C_VEL
LIN {X 0,Y 268.542,Z 458.876,A -85,B 0,C 180,E1 -17876.874,E2 -17876.874} C_VEL
LIN {X 0,Y 268.226,Z 459.93,A -85,B 0,C 180,E1 -17878.398,E2 -17878.398} C_VEL
LIN {X 0,Y 268.01,Z 460.531,A -85,B 0,C 180,E1 -17880.118,E2 -17880.118} C_VEL
LIN {X 0,Y 267.863,Z 460.489,A -85,B 0,C 180,E1 -17881.819,E2 -17881.819} C_VEL
LIN {X 0,Y 267.925,Z 459.815,A -85,B 0,C 180,E1 -17883.518,E2 -17883.518} C_VEL
LIN {X 0,Y 268.098,Z 458.512,A -85,B 0,C 180,E1 -17885.202,E2 -17885.202} C_VEL
LIN {X 0,Y 268.39,Z 456.568,A -85,B 0,C 180,E1 -17886.873,E2 -17886.873} C_VEL
LIN {X 0,Y 268.71,Z 453.955,A -85,B 0,C 180,E1 -17888.522,E2 -17888.522} C_VEL
LIN {X 0,Y 269.252,Z 449.602,A -85,B 0,C 180,E1 -17890.562,E2 -17890.562} C_VEL
LIN {X 0,Y 269.789,Z 445.262,A -85,B 0,C 180,E1 -17892.177,E2 -17892.177} C_VEL
LIN {X 0,Y 270.602,Z 439.355,A -85,B 0,C 180,E1 -17893.937,E2 -17893.937} C_VEL
LIN {X 0,Y 271.366,Z 433.477,A -85,B 0,C 180,E1 -17895.374,E2 -17895.374} C_VEL
LIN {X 0,Y 272.274,Z 426.662,A -85,B 0,C 180,E1 -17896.749,E2 -17896.749} C_VEL
LIN {X 0,Y 273.126,Z 419.735,A -85,B 0,C 180,E1 -17897.907,E2 -17897.907} C_VEL
LIN {X 0,Y 273.975,Z 412.501,A -85,B 0,C 180,E1 -17898.908,E2 -17898.908} C_VEL
LIN {X 0,Y 274.83,Z 403.828,A -85,B 0,C 180,E1 -17899.875,E2 -17899.875} C_VEL
LIN {X 0,Y 275.409,Z 395.136,A -85,B 0,C 180,E1 -17900.638,E2 -17900.638} C_VEL
LIN {X 0,Y 276.007,Z 385.359,A -85,B 0,C 180,E1 -17901.267,E2 -17901.267} C_VEL
LIN {X 0,Y 276.495,Z 374.778,A -85,B 0,C 180,E1 -17901.71,E2 -17901.71} C_VEL
LIN {X 0,Y 277.511,Z 329.791,A -85,B 0,C 180,E1 -17902.924,E2 -17902.924} C_VEL
LIN {X 0,Y 273.859,Z 309.731,A -85,B 0,C 180,E1 -17903.749,E2 -17903.749} C_VEL
LIN {X 0,Y 271.397,Z 301.396,A -85,B 0,C 180,E1 -17904.195,E2 -17904.195} C_VEL
LIN {X 0,Y 270.529,Z 296.603,A -85,B 0,C 180,E1 -17906.276,E2 -17906.276} C_VEL
LIN {X 0,Y 270.788,Z 296.568,A -85,B 0,C 180,E1 -17908.513,E2 -17908.513} C_VEL
LIN {X 0,Y 270.788,Z 296.567,A -85,B 0,C 180,E1 -17911.487,E2 -17911.487} C_VEL
LIN {X 0,Y 270.573,Z 296.591,A -85,B 0,C 180,E1 -17917.462,E2 -17917.462} C_VEL
LIN {X 0,Y 270.414,Z 296.612,A -85,B 0,C 180,E1 -17920.482,E2 -17920.482} C_VEL
LIN {X 0,Y 270.378,Z 296.616,A -85,B 0,C 180,E1 -17925.066,E2 -17925.066} C_VEL
LIN {X 0,Y 270.261,Z 296.626,A -85,B 0,C 180,E1 -17929.758,E2 -17929.758} C_VEL
LIN {X 0,Y 270.237,Z 296.633,A -85,B 0,C 180,E1 -17934.588,E2 -17934.588} C_VEL
LIN {X 0,Y 270.271,Z 296.63,A -85,B 0,C 180,E1 -17937.908,E2 -17937.908} C_VEL
LIN {X 0,Y 270.183,Z 296.64,A -85,B 0,C 180,E1 -17941.347,E2 -17941.347} C_VEL
LIN {X 0,Y 270.2,Z 296.639,A -85,B 0,C 180,E1 -17944.905,E2 -17944.905} C_VEL
LIN {X 0,Y 270.195,Z 296.639,A -85,B 0,C 180,E1 -17948.709,E2 -17948.709} C_VEL
LIN {X 0,Y 270.186,Z 296.637,A -85,B 0,C 180,E1 -17953.253,E2 -17953.253} C_VEL
LIN {X 0,Y 270.219,Z 296.638,A -85,B 0,C 180,E1 -17957.451,E2 -17957.451} C_VEL
LIN {X 0,Y 270.241,Z 296.633,A -85,B 0,C 180,E1 -17961.38,E2 -17961.38} C_VEL
LIN {X 0,Y 270.21,Z 296.628,A -85,B 0,C 180,E1 -17965.096,E2 -17965.096} C_VEL
LIN {X 0,Y 270.195,Z 296.636,A -85,B 0,C 180,E1 -17969.13,E2 -17969.13} C_VEL
LIN {X 0,Y 270.258,Z 296.635,A -85,B 0,C 180,E1 -17972.145,E2 -17972.145} C_VEL
LIN {X 0,Y 270.271,Z 296.626,A -85,B 0,C 180,E1 -17975.518,E2 -17975.518} C_VEL
LIN {X 0,Y 270.295,Z 296.619,A -85,B 0,C 180,E1 -17980.244,E2 -17980.244} C_VEL
LIN {X 0,Y 270.389,Z 296.616,A -85,B 0,C 180,E1 -17984.934,E2 -17984.934} C_VEL
LIN {X 0,Y 270.405,Z 296.611,A -85,B 0,C 180,E1 -17989.517,E2 -17989.517} C_VEL
LIN {X 0,Y 270.59,Z 296.588,A -85,B 0,C 180,E1 -17992.538,E2 -17992.538} C_VEL
LIN {X 0,Y 270.778,Z 296.563,A -85,B 0,C 180,E1 -17998.513,E2 -17998.513} C_VEL
LIN {X 0,Y 270.779,Z 296.567,A -85,B 0,C 180,E1 -18001.487,E2 -18001.487} C_VEL
LIN {X 0,Y 270.652,Z 296.581,A -85,B 0,C 180,E1 -18002.48,E2 -18002.48} C_VEL
LIN {X 0,Y 269.908,Z 296.677,A -85,B 0,C 180,E1 -18003.72,E2 -18003.72} C_VEL
LIN {X 0,Y 267,Z 297.035,A -85,B 0,C 180,E1 -18005.741,E2 -18005.741} C_VEL
LIN {X 0,Y 264.577,Z 297.336,A -85,B 0,C 180,E1 -18007.384,E2 -18007.384} C_VEL
LIN {X 0,Y 263.546,Z 297.46,A -85,B 0,C 180,E1 -18008.659,E2 -18008.659} C_VEL
LIN {X 0,Y 263.464,Z 297.472,A -85,B 0,C 180,E1 -18009.09,E2 -18009.09} C_VEL
LIN {X 0,Y 263.297,Z 297.499,A -85,B 0,C 180,E1 -18013.9,E2 -18013.9} C_VEL
LIN {X 0,Y 263.25,Z 297.504,A -85,B 0,C 180,E1 -18017.077,E2 -18017.077} C_VEL
LIN {X 0,Y 263.206,Z 297.503,A -85,B 0,C 180,E1 -18020.849,E2 -18020.849} C_VEL
LIN {X 0,Y 263.186,Z 297.511,A -85,B 0,C 180,E1 -18025.293,E2 -18025.293} C_VEL
LIN {X 0,Y 263.159,Z 297.513,A -85,B 0,C 180,E1 -18028.732,E2 -18028.732} C_VEL
LIN {X 0,Y 263.126,Z 297.522,A -85,B 0,C 180,E1 -18032.289,E2 -18032.289} C_VEL
LIN {X 0,Y 263.177,Z 297.513,A -85,B 0,C 180,E1 -18036.764,E2 -18036.764} C_VEL
LIN {X 0,Y 263.12,Z 297.511,A -85,B 0,C 180,E1 -18041.594,E2 -18041.594} C_VEL
LIN {X 0,Y 263.124,Z 297.519,A -85,B 0,C 180,E1 -18046.018,E2 -18046.018} C_VEL
LIN {X 0,Y 263.102,Z 297.522,A -85,B 0,C 180,E1 -18050.128,E2 -18050.128} C_VEL
LIN {X 0,Y 263.159,Z 297.515,A -85,B 0,C 180,E1 -18054.019,E2 -18054.019} C_VEL
LIN {X 0,Y 263.125,Z 297.521,A -85,B 0,C 180,E1 -18057.712,E2 -18057.712} C_VEL
LIN {X 0,Y 263.263,Z 297.707,A -85,B 0,C 180,E1 -18060.406,E2 -18060.406} C_VEL
LIN {X 0,Y 265.041,Z 307.408,A -85,B 0,C 180,E1 -18064.364,E2 -18064.364} C_VEL
LIN {X 0,Y 265.643,Z 311.026,A -85,B 0,C 180,E1 -18065.791,E2 -18065.791} C_VEL
LIN {X 0,Y 265.131,Z 315.351,A -85,B 0,C 180,E1 -18067.396,E2 -18067.396} C_VEL
LIN {X 0,Y 269.746,Z 349.153,A -85,B 0,C 180,E1 -18068.73,E2 -18068.73} C_VEL
LIN {X 0,Y 270.37,Z 355.514,A -85,B 0,C 180,E1 -18068.956,E2 -18068.956} C_VEL
LIN {X 0,Y 269.427,Z 392.619,A -85,B 0,C 180,E1 -18070.014,E2 -18070.014} C_VEL
LIN {X 0,Y 268.847,Z 402.411,A -85,B 0,C 180,E1 -18070.482,E2 -18070.482} C_VEL
LIN {X 0,Y 268.231,Z 409.766,A -85,B 0,C 180,E1 -18070.982,E2 -18070.982} C_VEL
LIN {X 0,Y 267.415,Z 419.071,A -85,B 0,C 180,E1 -18071.815,E2 -18071.815} C_VEL
LIN {X 0,Y 266.383,Z 428.655,A -85,B 0,C 180,E1 -18072.932,E2 -18072.932} C_VEL
LIN {X 0,Y 265.178,Z 438.443,A -85,B 0,C 180,E1 -18074.435,E2 -18074.435} C_VEL
LIN {X 0,Y 264.201,Z 445.347,A -85,B 0,C 180,E1 -18075.756,E2 -18075.756} C_VEL
LIN {X 0,Y 263.315,Z 451.882,A -85,B 0,C 180,E1 -18077.28,E2 -18077.28} C_VEL
LIN {X 0,Y 262.553,Z 457.308,A -85,B 0,C 180,E1 -18078.81,E2 -18078.81} C_VEL
LIN {X 0,Y 261.892,Z 462.8,A -85,B 0,C 180,E1 -18080.735,E2 -18080.735} C_VEL
LIN {X 0,Y 261.489,Z 466.363,A -85,B 0,C 180,E1 -18082.277,E2 -18082.277} C_VEL
LIN {X 0,Y 261.259,Z 469.279,A -85,B 0,C 180,E1 -18083.823,E2 -18083.823} C_VEL
LIN {X 0,Y 261.099,Z 471.577,A -85,B 0,C 180,E1 -18085.368,E2 -18085.368} C_VEL
LIN {X 0,Y 261.11,Z 473.237,A -85,B 0,C 180,E1 -18086.914,E2 -18086.914} C_VEL
LIN {X 0,Y 261.114,Z 474.365,A -85,B 0,C 180,E1 -18088.458,E2 -18088.458} C_VEL
LIN {X 0,Y 261.125,Z 475.008,A -85,B 0,C 180,E1 -18090,E2 -18090} C_VEL
LIN {X 0,Y 261.089,Z 475.18,A -85,B 0,C 180,E1 -18091.542,E2 -18091.542} C_VEL
LIN {X 0,Y 261.077,Z 474.821,A -85,B 0,C 180,E1 -18093.086,E2 -18093.086} C_VEL
LIN {X 0,Y 261.13,Z 473.445,A -85,B 0,C 180,E1 -18095.249,E2 -18095.249} C_VEL
LIN {X 0,Y 261.762,Z 469.377,A -85,B 0,C 180,E1 -18098.492,E2 -18098.492} C_VEL
LIN {X 0,Y 262.599,Z 465.001,A -85,B 0,C 180,E1 -18100.797,E2 -18100.797} C_VEL
LIN {X 0,Y 263.815,Z 458.961,A -85,B 0,C 180,E1 -18103.087,E2 -18103.087} C_VEL
LIN {X 0,Y 264.9,Z 453.979,A -85,B 0,C 180,E1 -18104.598,E2 -18104.598} C_VEL
LIN {X 0,Y 266.103,Z 447.991,A -85,B 0,C 180,E1 -18106.099,E2 -18106.099} C_VEL
LIN {X 0,Y 267.572,Z 440.718,A -85,B 0,C 180,E1 -18107.581,E2 -18107.581} C_VEL
LIN {X 0,Y 268.761,Z 434.195,A -85,B 0,C 180,E1 -18108.682,E2 -18108.682} C_VEL
LIN {X 0,Y 270.125,Z 426.318,A -85,B 0,C 180,E1 -18109.768,E2 -18109.768} C_VEL
LIN {X 0,Y 271.113,Z 418.269,A -85,B 0,C 180,E1 -18110.682,E2 -18110.682} C_VEL
LIN {X 0,Y 272.328,Z 408.828,A -85,B 0,C 180,E1 -18111.491,E2 -18111.491} C_VEL
LIN {X 0,Y 273.279,Z 399.293,A -85,B 0,C 180,E1 -18112.086,E2 -18112.086} C_VEL
LIN {X 0,Y 273.945,Z 388.174,A -85,B 0,C 180,E1 -18112.546,E2 -18112.546} C_VEL
LIN {X 0,Y 274.8,Z 355.274,A -85,B 0,C 180,E1 -18113.471,E2 -18113.471} C_VEL
LIN {X 0,Y 272.441,Z 338.403,A -85,B 0,C 180,E1 -18114.257,E2 -18114.257} C_VEL
LIN {X 0,Y 268.779,Z 320.009,A -85,B 0,C 180,E1 -18115.268,E2 -18115.268} C_VEL
LIN {X 0,Y 266.639,Z 314.018,A -85,B 0,C 180,E1 -18115.756,E2 -18115.756} C_VEL
LIN {X 0,Y 264.883,Z 304.99,A -85,B 0,C 180,E1 -18119.507,E2 -18119.507} C_VEL
LIN {X 0,Y 263.157,Z 297.52,A -85,B 0,C 180,E1 -18122.851,E2 -18122.851} C_VEL
LIN {X 0,Y 263.179,Z 297.517,A -85,B 0,C 180,E1 -18126.762,E2 -18126.762} C_VEL
LIN {X 0,Y 263.12,Z 297.525,A -85,B 0,C 180,E1 -18131.593,E2 -18131.593} C_VEL
LIN {X 0,Y 263.1,Z 297.527,A -85,B 0,C 180,E1 -18136.154,E2 -18136.154} C_VEL
LIN {X 0,Y 263.1,Z 297.525,A -85,B 0,C 180,E1 -18140.127,E2 -18140.127} C_VEL
LIN {X 0,Y 263.169,Z 297.513,A -85,B 0,C 180,E1 -18144.019,E2 -18144.019} C_VEL
LIN {X 0,Y 263.126,Z 297.51,A -85,B 0,C 180,E1 -18147.711,E2 -18147.711} C_VEL
LIN {X 0,Y 263.194,Z 297.501,A -85,B 0,C 180,E1 -18151.783,E2 -18151.783} C_VEL
LIN {X 0,Y 263.194,Z 297.511,A -85,B 0,C 180,E1 -18155.212,E2 -18155.212} C_VEL
LIN {X 0,Y 263.255,Z 297.496,A -85,B 0,C 180,E1 -18159.693,E2 -18159.693} C_VEL
LIN {X 0,Y 263.337,Z 297.478,A -85,B 0,C 180,E1 -18164.521,E2 -18164.521} C_VEL
LIN {X 0,Y 263.347,Z 297.485,A -85,B 0,C 180,E1 -18169.233,E2 -18169.233} C_VEL
LIN {X 0,Y 263.55,Z 297.459,A -85,B 0,C 180,E1 -18172.338,E2 -18172.338} C_VEL
LIN {X 0,Y 263.742,Z 297.437,A -85,B 0,C 180,E1 -18178.473,E2 -18178.473} C_VEL
LIN {X 0,Y 263.741,Z 297.431,A -85,B 0,C 180,E1 -18181.527,E2 -18181.527} C_VEL
LIN {X 0,Y 263.52,Z 297.46,A -85,B 0,C 180,E1 -18187.663,E2 -18187.663} C_VEL
LIN {X 0,Y 263.346,Z 297.494,A -85,B 0,C 180,E1 -18190.767,E2 -18190.767} C_VEL
LIN {X 0,Y 263.337,Z 297.494,A -85,B 0,C 180,E1 -18195.479,E2 -18195.479} C_VEL
LIN {X 0,Y 263.257,Z 297.501,A -85,B 0,C 180,E1 -18200.307,E2 -18200.307} C_VEL
LIN {X 0,Y 263.202,Z 297.515,A -85,B 0,C 180,E1 -18205.292,E2 -18205.292} C_VEL
LIN {X 0,Y 263.161,Z 297.514,A -85,B 0,C 180,E1 -18208.732,E2 -18208.732} C_VEL
LIN {X 0,Y 263.162,Z 297.518,A -85,B 0,C 180,E1 -18213.194,E2 -18213.194} C_VEL
LIN {X 0,Y 263.196,Z 297.644,A -85,B 0,C 180,E1 -18214.131,E2 -18214.131} C_VEL
LIN {X 0,Y 264.254,Z 301.98,A -85,B 0,C 180,E1 -18216.031,E2 -18216.031} C_VEL
LIN {X 0,Y 271.247,Z 317.463,A -85,B 0,C 180,E1 -18217.392,E2 -18217.392} C_VEL
LIN {X 0,Y 273.995,Z 324.685,A -85,B 0,C 180,E1 -18217.938,E2 -18217.938} C_VEL
LIN {X 0,Y 275.566,Z 333.77,A -85,B 0,C 180,E1 -18218.397,E2 -18218.397} C_VEL
LIN {X 0,Y 274.038,Z 378.154,A -85,B 0,C 180,E1 -18219.643,E2 -18219.643} C_VEL
LIN {X 0,Y 273.431,Z 387.748,A -85,B 0,C 180,E1 -18220.088,E2 -18220.088} C_VEL
LIN {X 0,Y 272.628,Z 397.73,A -85,B 0,C 180,E1 -18220.78,E2 -18220.78} C_VEL
LIN {X 0,Y 271.273,Z 409.13,A -85,B 0,C 180,E1 -18221.88,E2 -18221.88} C_VEL
LIN {X 0,Y 269.982,Z 417.777,A -85,B 0,C 180,E1 -18222.997,E2 -18222.997} C_VEL
LIN {X 0,Y 268.66,Z 425.65,A -85,B 0,C 180,E1 -18224.267,E2 -18224.267} C_VEL
LIN {X 0,Y 267.449,Z 431.791,A -85,B 0,C 180,E1 -18225.457,E2 -18225.457} C_VEL
LIN {X 0,Y 266.084,Z 438.353,A -85,B 0,C 180,E1 -18227.007,E2 -18227.007} C_VEL
LIN {X 0,Y 265.004,Z 443.458,A -85,B 0,C 180,E1 -18228.472,E2 -18228.472} C_VEL
LIN {X 0,Y 263.854,Z 448.544,A -85,B 0,C 180,E1 -18230.265,E2 -18230.265} C_VEL
LIN {X 0,Y 262.982,Z 452.607,A -85,B 0,C 180,E1 -18232.074,E2 -18232.074} C_VEL
LIN {X 0,Y 262.171,Z 455.737,A -85,B 0,C 180,E1 -18233.862,E2 -18233.862} C_VEL
LIN {X 0,Y 261.752,Z 458.084,A -85,B 0,C 180,E1 -18235.679,E2 -18235.679} C_VEL
LIN {X 0,Y 261.303,Z 459.676,A -85,B 0,C 180,E1 -18237.459,E2 -18237.459} C_VEL
LIN {X 0,Y 260.976,Z 460.642,A -85,B 0,C 180,E1 -18239.514,E2 -18239.514} C_VEL
LIN {X 0,Y 260.813,Z 460.85,A -85,B 0,C 180,E1 -18240.986,E2 -18240.986} C_VEL
LIN {X 0,Y 260.795,Z 460.424,A -85,B 0,C 180,E1 -18242.785,E2 -18242.785} C_VEL
LIN {X 0,Y 260.898,Z 459.37,A -85,B 0,C 180,E1 -18244.47,E2 -18244.47} C_VEL
LIN {X 0,Y 261.334,Z 456.559,A -85,B 0,C 180,E1 -18247.05,E2 -18247.05} C_VEL
LIN {X 0,Y 261.663,Z 453.899,A -85,B 0,C 180,E1 -18248.741,E2 -18248.741} C_VEL
LIN {X 0,Y 262.142,Z 450.14,A -85,B 0,C 180,E1 -18250.567,E2 -18250.567} C_VEL
LIN {X 0,Y 262.789,Z 445.057,A -85,B 0,C 180,E1 -18252.491,E2 -18252.491} C_VEL
LIN {X 0,Y 263.61,Z 439.449,A -85,B 0,C 180,E1 -18254.193,E2 -18254.193} C_VEL
LIN {X 0,Y 264.479,Z 433.078,A -85,B 0,C 180,E1 -18255.771,E2 -18255.771} C_VEL
LIN {X 0,Y 265.432,Z 426.1,A -85,B 0,C 180,E1 -18257.189,E2 -18257.189} C_VEL
LIN {X 0,Y 266.351,Z 418.897,A -85,B 0,C 180,E1 -18258.394,E2 -18258.394} C_VEL
LIN {X 0,Y 267.201,Z 411.666,A -85,B 0,C 180,E1 -18259.391,E2 -18259.391} C_VEL
LIN {X 0,Y 268.073,Z 402.763,A -85,B 0,C 180,E1 -18260.379,E2 -18260.379} C_VEL
LIN {X 0,Y 268.771,Z 393.071,A -85,B 0,C 180,E1 -18261.207,E2 -18261.207} C_VEL
LIN {X 0,Y 269.515,Z 380.806,A -85,B 0,C 180,E1 -18261.918,E2 -18261.918} C_VEL
LIN {X 0,Y 270.075,Z 361.058,A -85,B 0,C 180,E1 -18262.524,E2 -18262.524} C_VEL
LIN {X 0,Y 270.694,Z 330.102,A -85,B 0,C 180,E1 -18263.38,E2 -18263.38} C_VEL
LIN {X 0,Y 267.336,Z 311.736,A -85,B 0,C 180,E1 -18264.154,E2 -18264.154} C_VEL
LIN {X 0,Y 264.199,Z 301.628,A -85,B 0,C 180,E1 -18264.706,E2 -18264.706} C_VEL
LIN {X 0,Y 263.531,Z 297.475,A -85,B 0,C 180,E1 -18266.56,E2 -18266.56} C_VEL
LIN {X 0,Y 263.805,Z 297.44,A -85,B 0,C 180,E1 -18270,E2 -18270} C_VEL
LIN {X 0,Y 263.563,Z 297.464,A -85,B 0,C 180,E1 -18273.057,E2 -18273.057} C_VEL
LIN {X 0,Y 263.535,Z 297.468,A -85,B 0,C 180,E1 -18277.662,E2 -18277.662} C_VEL
LIN {X 0,Y 263.356,Z 297.489,A -85,B 0,C 180,E1 -18280.766,E2 -18280.766} C_VEL
LIN {X 0,Y 263.324,Z 297.494,A -85,B 0,C 180,E1 -18285.479,E2 -18285.479} C_VEL
LIN {X 0,Y 263.238,Z 297.502,A -85,B 0,C 180,E1 -18290.308,E2 -18290.308} C_VEL
LIN {X 0,Y 263.192,Z 297.512,A -85,B 0,C 180,E1 -18295.292,E2 -18295.292} C_VEL
LIN {X 0,Y 263.179,Z 297.517,A -85,B 0,C 180,E1 -18298.729,E2 -18298.729} C_VEL
LIN {X 0,Y 263.132,Z 297.516,A -85,B 0,C 180,E1 -18302.287,E2 -18302.287} C_VEL
LIN {X 0,Y 263.179,Z 297.514,A -85,B 0,C 180,E1 -18306.762,E2 -18306.762} C_VEL
LIN {X 0,Y 263.127,Z 297.516,A -85,B 0,C 180,E1 -18311.594,E2 -18311.594} C_VEL
LIN {X 0,Y 263.142,Z 297.517,A -85,B 0,C 180,E1 -18316.02,E2 -18316.02} C_VEL
LIN {X 0,Y 263.156,Z 297.515,A -85,B 0,C 180,E1 -18320.136,E2 -18320.136} C_VEL
LIN {X 0,Y 263.183,Z 297.506,A -85,B 0,C 180,E1 -18324.021,E2 -18324.021} C_VEL
LIN {X 0,Y 263.128,Z 297.517,A -85,B 0,C 180,E1 -18327.711,E2 -18327.711} C_VEL
LIN {X 0,Y 263.193,Z 297.512,A -85,B 0,C 180,E1 -18331.783,E2 -18331.783} C_VEL
LIN {X 0,Y 263.22,Z 297.504,A -85,B 0,C 180,E1 -18335.2,E2 -18335.2} C_VEL
LIN {X 0,Y 263.257,Z 297.491,A -85,B 0,C 180,E1 -18339.693,E2 -18339.693} C_VEL
LIN {X 0,Y 263.337,Z 297.495,A -85,B 0,C 180,E1 -18344.521,E2 -18344.521} C_VEL
LIN {X 0,Y 263.347,Z 297.491,A -85,B 0,C 180,E1 -18349.233,E2 -18349.233} C_VEL
LIN {X 0,Y 263.55,Z 297.463,A -85,B 0,C 180,E1 -18352.338,E2 -18352.338} C_VEL
LIN {X 0,Y 263.742,Z 297.438,A -85,B 0,C 180,E1 -18358.473,E2 -18358.473} C_VEL
LIN {X 0,Y 263.743,Z 297.444,A -85,B 0,C 180,E1 -18361.527,E2 -18361.527} C_VEL
LIN {X 0,Y 263.55,Z 297.462,A -85,B 0,C 180,E1 -18367.662,E2 -18367.662} C_VEL
LIN {X 0,Y 263.464,Z 297.472,A -85,B 0,C 180,E1 -18369.09,E2 -18369.09} C_VEL
LIN {X 0,Y 262.77,Z 297.563,A -85,B 0,C 180,E1 -18370.365,E2 -18370.365} C_VEL
LIN {X 0,Y 259.808,Z 297.93,A -85,B 0,C 180,E1 -18372.438,E2 -18372.438} C_VEL
LIN {X 0,Y 257.331,Z 298.241,A -85,B 0,C 180,E1 -18374.125,E2 -18374.125} C_VEL
LIN {X 0,Y 256.322,Z 298.369,A -85,B 0,C 180,E1 -18375.436,E2 -18375.436} C_VEL
LIN {X 0,Y 256.27,Z 298.375,A -85,B 0,C 180,E1 -18375.88,E2 -18375.88} C_VEL
LIN {X 0,Y 256.177,Z 298.383,A -85,B 0,C 180,E1 -18379.221,E2 -18379.221} C_VEL
LIN {X 0,Y 256.076,Z 298.394,A -85,B 0,C 180,E1 -18382.596,E2 -18382.596} C_VEL
LIN {X 0,Y 256.122,Z 298.396,A -85,B 0,C 180,E1 -18386.042,E2 -18386.042} C_VEL
LIN {X 0,Y 256.097,Z 298.393,A -85,B 0,C 180,E1 -18389.602,E2 -18389.602} C_VEL
LIN {X 0,Y 256.062,Z 298.399,A -85,B 0,C 180,E1 -18393.293,E2 -18393.293} C_VEL
LIN {X 0,Y 256.109,Z 298.391,A -85,B 0,C 180,E1 -18397.271,E2 -18397.271} C_VEL
LIN {X 0,Y 256.05,Z 298.392,A -85,B 0,C 180,E1 -18401.204,E2 -18401.204} C_VEL
LIN {X 0,Y 256.058,Z 298.399,A -85,B 0,C 180,E1 -18405.53,E2 -18405.53} C_VEL
LIN {X 0,Y 256.051,Z 298.405,A -85,B 0,C 180,E1 -18408.797,E2 -18408.797} C_VEL
LIN {X 0,Y 256.126,Z 298.394,A -85,B 0,C 180,E1 -18412.868,E2 -18412.868} C_VEL
LIN {X 0,Y 256.063,Z 298.4,A -85,B 0,C 180,E1 -18416.708,E2 -18416.708} C_VEL
LIN {X 0,Y 256.18,Z 298.548,A -85,B 0,C 180,E1 -18420.07,E2 -18420.07} C_VEL
LIN {X 0,Y 257.983,Z 308.289,A -85,B 0,C 180,E1 -18424.16,E2 -18424.16} C_VEL
LIN {X 0,Y 258.629,Z 312.713,A -85,B 0,C 180,E1 -18425.946,E2 -18425.946} C_VEL
LIN {X 0,Y 258.288,Z 315.2,A -85,B 0,C 180,E1 -18426.891,E2 -18426.891} C_VEL
LIN {X 0,Y 263.188,Z 351.979,A -85,B 0,C 180,E1 -18428.367,E2 -18428.367} C_VEL
LIN {X 0,Y 263.564,Z 357.246,A -85,B 0,C 180,E1 -18428.55,E2 -18428.55} C_VEL
LIN {X 0,Y 262.614,Z 392.849,A -85,B 0,C 180,E1 -18429.597,E2 -18429.597} C_VEL
LIN {X 0,Y 261.983,Z 402.953,A -85,B 0,C 180,E1 -18430.102,E2 -18430.102} C_VEL
LIN {X 0,Y 261.242,Z 411.922,A -85,B 0,C 180,E1 -18430.759,E2 -18430.759} C_VEL
LIN {X 0,Y 260.064,Z 423.147,A -85,B 0,C 180,E1 -18431.894,E2 -18431.894} C_VEL
LIN {X 0,Y 259.056,Z 431.701,A -85,B 0,C 180,E1 -18433.044,E2 -18433.044} C_VEL
LIN {X 0,Y 257.99,Z 439.765,A -85,B 0,C 180,E1 -18434.395,E2 -18434.395} C_VEL
LIN {X 0,Y 257.029,Z 446.422,A -85,B 0,C 180,E1 -18435.754,E2 -18435.754} C_VEL
LIN {X 0,Y 256.154,Z 452.749,A -85,B 0,C 180,E1 -18437.321,E2 -18437.321} C_VEL
LIN {X 0,Y 255.411,Z 457.992,A -85,B 0,C 180,E1 -18438.895,E2 -18438.895} C_VEL
LIN {X 0,Y 254.861,Z 462.356,A -85,B 0,C 180,E1 -18440.477,E2 -18440.477} C_VEL
LIN {X 0,Y 254.284,Z 467.503,A -85,B 0,C 180,E1 -18442.856,E2 -18442.856} C_VEL
LIN {X 0,Y 254.012,Z 471.248,A -85,B 0,C 180,E1 -18445.239,E2 -18445.239} C_VEL
LIN {X 0,Y 254.007,Z 472.935,A -85,B 0,C 180,E1 -18446.828,E2 -18446.828} C_VEL
LIN {X 0,Y 254.022,Z 474.105,A -85,B 0,C 180,E1 -18448.415,E2 -18448.415} C_VEL
LIN {X 0,Y 254.052,Z 474.791,A -85,B 0,C 180,E1 -18450,E2 -18450} C_VEL
LIN {X 0,Y 253.997,Z 475.002,A -85,B 0,C 180,E1 -18451.585,E2 -18451.585} C_VEL
LIN {X 0,Y 253.977,Z 474.648,A -85,B 0,C 180,E1 -18453.172,E2 -18453.172} C_VEL
LIN {X 0,Y 254.052,Z 473.472,A -85,B 0,C 180,E1 -18455.199,E2 -18455.199} C_VEL
LIN {X 0,Y 254.517,Z 470.501,A -85,B 0,C 180,E1 -18457.936,E2 -18457.936} C_VEL
LIN {X 0,Y 254.999,Z 468.088,A -85,B 0,C 180,E1 -18459.518,E2 -18459.518} C_VEL
LIN {X 0,Y 255.968,Z 463.163,A -85,B 0,C 180,E1 -18461.883,E2 -18461.883} C_VEL
LIN {X 0,Y 257.19,Z 457.882,A -85,B 0,C 180,E1 -18463.833,E2 -18463.833} C_VEL
LIN {X 0,Y 258.301,Z 452.72,A -85,B 0,C 180,E1 -18465.383,E2 -18465.383} C_VEL
LIN {X 0,Y 259.605,Z 446.521,A -85,B 0,C 180,E1 -18466.919,E2 -18466.919} C_VEL
LIN {X 0,Y 261.032,Z 440.023,A -85,B 0,C 180,E1 -18468.239,E2 -18468.239} C_VEL
LIN {X 0,Y 262.527,Z 432.188,A -85,B 0,C 180,E1 -18469.55,E2 -18469.55} C_VEL
LIN {X 0,Y 263.906,Z 423.947,A -85,B 0,C 180,E1 -18470.661,E2 -18470.661} C_VEL
LIN {X 0,Y 265.318,Z 413.523,A -85,B 0,C 180,E1 -18471.767,E2 -18471.767} C_VEL
LIN {X 0,Y 266.629,Z 402.376,A -85,B 0,C 180,E1 -18472.576,E2 -18472.576} C_VEL
LIN {X 0,Y 267.356,Z 393.002,A -85,B 0,C 180,E1 -18473.043,E2 -18473.043} C_VEL
LIN {X 0,Y 268.443,Z 363.062,A -85,B 0,C 180,E1 -18473.931,E2 -18473.931} C_VEL
LIN {X 0,Y 268.427,Z 355.371,A -85,B 0,C 180,E1 -18474.177,E2 -18474.177} C_VEL
LIN {X 0,Y 266.143,Z 339.244,A -85,B 0,C 180,E1 -18474.964,E2 -18474.964} C_VEL
LIN {X 0,Y 262.691,Z 322.01,A -85,B 0,C 180,E1 -18475.953,E2 -18475.953} C_VEL
LIN {X 0,Y 259.398,Z 313.795,A -85,B 0,C 180,E1 -18476.687,E2 -18476.687} C_VEL
LIN {X 0,Y 257.754,Z 305.48,A -85,B 0,C 180,E1 -18480.291,E2 -18480.291} C_VEL
LIN {X 0,Y 256.104,Z 298.396,A -85,B 0,C 180,E1 -18483.615,E2 -18483.615} C_VEL
LIN {X 0,Y 256.111,Z 298.398,A -85,B 0,C 180,E1 -18487.27,E2 -18487.27} C_VEL
LIN {X 0,Y 256.051,Z 298.409,A -85,B 0,C 180,E1 -18491.203,E2 -18491.203} C_VEL
LIN {X 0,Y 256.036,Z 298.404,A -85,B 0,C 180,E1 -18495.533,E2 -18495.533} C_VEL
LIN {X 0,Y 256.049,Z 298.397,A -85,B 0,C 180,E1 -18498.796,E2 -18498.796} C_VEL
LIN {X 0,Y 256.131,Z 298.383,A -85,B 0,C 180,E1 -18502.868,E2 -18502.868} C_VEL
LIN {X 0,Y 256.062,Z 298.393,A -85,B 0,C 180,E1 -18506.707,E2 -18506.707} C_VEL
LIN {X 0,Y 256.108,Z 298.394,A -85,B 0,C 180,E1 -18510.4,E2 -18510.4} C_VEL
LIN {X 0,Y 256.164,Z 298.387,A -85,B 0,C 180,E1 -18514.87,E2 -18514.87} C_VEL
LIN {X 0,Y 256.155,Z 298.377,A -85,B 0,C 180,E1 -18519.104,E2 -18519.104} C_VEL
LIN {X 0,Y 256.287,Z 298.357,A -85,B 0,C 180,E1 -18524.084,E2 -18524.084} C_VEL
LIN {X 0,Y 256.285,Z 298.372,A -85,B 0,C 180,E1 -18527.328,E2 -18527.328} C_VEL
LIN {X 0,Y 256.507,Z 298.335,A -85,B 0,C 180,E1 -18532.126,E2 -18532.126} C_VEL
LIN {X 0,Y 256.486,Z 298.331,A -85,B 0,C 180,E1 -18536.859,E2 -18536.859} C_VEL
LIN {X 0,Y 256.756,Z 298.311,A -85,B 0,C 180,E1 -18540,E2 -18540} C_VEL
LIN {X 0,Y 256.484,Z 298.335,A -85,B 0,C 180,E1 -18543.142,E2 -18543.142} C_VEL
LIN {X 0,Y 256.462,Z 298.339,A -85,B 0,C 180,E1 -18547.876,E2 -18547.876} C_VEL
LIN {X 0,Y 256.289,Z 298.37,A -85,B 0,C 180,E1 -18551.067,E2 -18551.067} C_VEL
LIN {X 0,Y 256.244,Z 298.379,A -85,B 0,C 180,E1 -18554.291,E2 -18554.291} C_VEL
LIN {X 0,Y 256.197,Z 298.381,A -85,B 0,C 180,E1 -18557.563,E2 -18557.563} C_VEL
